gfCNCPoint4[19231] = {X 485.1607, Y 22.5274, Z -6.3333, A 0.000, B 0.000, C 0.000 }
gfCNCPoint4[19232] = {X 489.1455, Y 22.8760, Z -6.3333, A 0.000, B 0.000, C 0.000 }
gfCNCPoint4[19233] = {X 493.6890, Y 22.8760, Z -6.3333, A 0.000, B 0.000, C 0.000 }
gfCNCPoint4[19234] = {X 493.6890, Y 19.4624, Z -6.3333, A 0.000, B 0.000, C 0.000 }
gfCNCPoint4[19235] = {X 487.6634, Y 19.4617, Z -6.3333, A 0.000, B 0.000, C 0.000 }
gfCNCPoint4[19236] = {X 486.9708, Y 19.4665, Z -6.3333, A 0.000, B 0.000, C 0.000 }
gfCNCPoint4[19237] = {X 485.8326, Y 19.5401, Z -6.3333, A 0.000, B 0.000, C 0.000 }
gfCNCPoint4[19238] = {X 484.7145, Y 19.7657, Z -6.3333, A 0.000, B 0.000, C 0.000 }
gfCNCPoint4[19239] = {X 484.4483, Y 19.9152, Z -6.3333, A 0.000, B 0.000, C 0.000 }
gfCNCPoint4[19240] = {X 484.2838, Y 20.1725, Z -6.3333, A 0.000, B 0.000, C 0.000 }
gfCNCPoint4[19241] = {X 484.1061, Y 20.9736, Z -6.3333, A 0.000, B 0.000, C 0.000 }
gfCNCPoint4[19242] = {X 484.1000, Y 21.7941, Z -6.3333, A 0.000, B 0.000, C 0.000 }
gfCNCPoint4[19243] = {X 484.2657, Y 22.5977, Z -6.3333, A 0.000, B 0.000, C 0.000 }
gfCNCPoint4[19244] = {X 484.5770, Y 22.7005, Z -6.3333, A 0.000, B 0.000, C 0.000 }
gfCNCPoint4[19245] = {X 484.9007, Y 22.7530, Z -6.3333, A 0.000, B 0.000, C 0.000 }
gfCNCPoint4[19246] = {X 486.2706, Y 22.8551, Z -6.3333, A 0.000, B 0.000, C 0.000 }
gfCNCPoint4[19247] = {X 487.6442, Y 22.8760, Z -6.3333, A 0.000, B 0.000, C 0.000 }
gfCNCPoint4[19248] = {X 489.1455, Y 22.8760, Z -6.3333, A 0.000, B 0.000, C 0.000 }
gfCNCPoint4[19249] = {X 493.1302, Y 22.5274, Z -6.3333, A 0.000, B 0.000, C 0.000 }
gfCNCPoint4[19250] = {X 485.1607, Y 22.6074, Z -6.3333, A 0.000, B 0.000, C 0.000 }
gfCNCPoint4[19251] = {X 489.1455, Y 22.9560, Z -6.3333, A 0.000, B 0.000, C 0.000 }
gfCNCPoint4[19252] = {X 493.7690, Y 22.9560, Z -6.3333, A 0.000, B 0.000, C 0.000 }
gfCNCPoint4[19253] = {X 493.7690, Y 19.3824, Z -6.3333, A 0.000, B 0.000, C 0.000 }
gfCNCPoint4[19254] = {X 487.6632, Y 19.3817, Z -6.3333, A 0.000, B 0.000, C 0.000 }
gfCNCPoint4[19255] = {X 486.9707, Y 19.3865, Z -6.3333, A 0.000, B 0.000, C 0.000 }
gfCNCPoint4[19256] = {X 485.8219, Y 19.4608, Z -6.3333, A 0.000, B 0.000, C 0.000 }
gfCNCPoint4[19257] = {X 484.6935, Y 19.6886, Z -6.3333, A 0.000, B 0.000, C 0.000 }
gfCNCPoint4[19258] = {X 484.3933, Y 19.8571, Z -6.3333, A 0.000, B 0.000, C 0.000 }
gfCNCPoint4[19259] = {X 484.2079, Y 20.1470, Z -6.3333, A 0.000, B 0.000, C 0.000 }
gfCNCPoint4[19260] = {X 484.0252, Y 20.9767, Z -6.3333, A 0.000, B 0.000, C 0.000 }
gfCNCPoint4[19261] = {X 484.0228, Y 21.8262, Z -6.3333, A 0.000, B 0.000, C 0.000 }
gfCNCPoint4[19262] = {X 484.2007, Y 22.6569, Z -6.3333, A 0.000, B 0.000, C 0.000 }
gfCNCPoint4[19263] = {X 484.5397, Y 22.7736, Z -6.3333, A 0.000, B 0.000, C 0.000 }
gfCNCPoint4[19264] = {X 484.8932, Y 22.8327, Z -6.3333, A 0.000, B 0.000, C 0.000 }
gfCNCPoint4[19265] = {X 486.2672, Y 22.9351, Z -6.3333, A 0.000, B 0.000, C 0.000 }
gfCNCPoint4[19266] = {X 487.6448, Y 22.9560, Z -6.3333, A 0.000, B 0.000, C 0.000 }
gfCNCPoint4[19267] = {X 489.1455, Y 22.9560, Z -6.3333, A 0.000, B 0.000, C 0.000 }
gfCNCPoint4[19268] = {X 493.1302, Y 22.6074, Z -6.3333, A 0.000, B 0.000, C 0.000 }
gfCNCPoint4[19269] = {X 493.1302, Y 22.6074, Z -3.3333, A 0.000, B 0.000, C 0.000 }
gfCNCPoint4[19270] = {X 493.1302, Y 22.6074, Z 11.0000, A 0.000, B 0.000, C 0.000 }
gfCNCPoint4[19271] = {X 448.7147, Y 19.7824, Z 11.0000, A 0.000, B 0.000, C 0.000 }
gfCNCPoint4[19272] = {X 448.7147, Y 19.7824, Z -2.5000, A 0.000, B 0.000, C 0.000 }
gfCNCPoint4[19273] = {X 444.0414, Y 19.7824, Z -3.7522, A 0.000, B 0.000, C 0.000 }
gfCNCPoint4[19274] = {X 443.3486, Y 19.7986, Z -3.9379, A 0.000, B 0.000, C 0.000 }
gfCNCPoint4[19275] = {X 442.7492, Y 19.8053, Z -4.0985, A 0.000, B 0.000, C 0.000 }
gfCNCPoint4[19276] = {X 442.0368, Y 19.9286, Z -4.2922, A 0.000, B 0.000, C 0.000 }
gfCNCPoint4[19277] = {X 441.4699, Y 20.1238, Z -4.4529, A 0.000, B 0.000, C 0.000 }
gfCNCPoint4[19278] = {X 441.3670, Y 20.1592, Z -4.4820, A 0.000, B 0.000, C 0.000 }
gfCNCPoint4[19279] = {X 441.1893, Y 20.7188, Z -4.6394, A 0.000, B 0.000, C 0.000 }
gfCNCPoint4[19280] = {X 441.1557, Y 21.8876, Z -4.9527, A 0.000, B 0.000, C 0.000 }
gfCNCPoint4[19281] = {X 441.2739, Y 22.3510, Z -5.0808, A 0.000, B 0.000, C 0.000 }
gfCNCPoint4[19282] = {X 441.5039, Y 22.4262, Z -5.1457, A 0.000, B 0.000, C 0.000 }
gfCNCPoint4[19283] = {X 441.7450, Y 22.4480, Z -5.2105, A 0.000, B 0.000, C 0.000 }
gfCNCPoint4[19284] = {X 443.0096, Y 22.5623, Z -5.5508, A 0.000, B 0.000, C 0.000 }
gfCNCPoint4[19285] = {X 443.1211, Y 22.5669, Z -5.5807, A 0.000, B 0.000, C 0.000 }
gfCNCPoint4[19286] = {X 444.3942, Y 22.5560, Z -5.9218, A 0.000, B 0.000, C 0.000 }
gfCNCPoint4[19287] = {X 445.9301, Y 22.5560, Z -6.3333, A 0.000, B 0.000, C 0.000 }
gfCNCPoint4[19288] = {X 450.1184, Y 22.5560, Z -6.3333, A 0.000, B 0.000, C 0.000 }
gfCNCPoint4[19289] = {X 450.1184, Y 19.7824, Z -6.3333, A 0.000, B 0.000, C 0.000 }
gfCNCPoint4[19290] = {X 444.0414, Y 19.7824, Z -6.3333, A 0.000, B 0.000, C 0.000 }
gfCNCPoint4[19291] = {X 443.3486, Y 19.7986, Z -6.3333, A 0.000, B 0.000, C 0.000 }
gfCNCPoint4[19292] = {X 442.3962, Y 19.8858, Z -6.3333, A 0.000, B 0.000, C 0.000 }
gfCNCPoint4[19293] = {X 441.4699, Y 20.1238, Z -6.3333, A 0.000, B 0.000, C 0.000 }
gfCNCPoint4[19294] = {X 441.3855, Y 20.1772, Z -6.3333, A 0.000, B 0.000, C 0.000 }
gfCNCPoint4[19295] = {X 441.3341, Y 20.2630, Z -6.3333, A 0.000, B 0.000, C 0.000 }
gfCNCPoint4[19296] = {X 441.1841, Y 20.9512, Z -6.3333, A 0.000, B 0.000, C 0.000 }
gfCNCPoint4[19297] = {X 441.1638, Y 21.6553, Z -6.3333, A 0.000, B 0.000, C 0.000 }
gfCNCPoint4[19298] = {X 441.2739, Y 22.3510, Z -6.3333, A 0.000, B 0.000, C 0.000 }
gfCNCPoint4[19299] = {X 441.5067, Y 22.4128, Z -6.3333, A 0.000, B 0.000, C 0.000 }
gfCNCPoint4[19300] = {X 441.7450, Y 22.4480, Z -6.3333, A 0.000, B 0.000, C 0.000 }
gfCNCPoint4[19301] = {X 443.0683, Y 22.5347, Z -6.3333, A 0.000, B 0.000, C 0.000 }
gfCNCPoint4[19302] = {X 444.3942, Y 22.5560, Z -6.3333, A 0.000, B 0.000, C 0.000 }
gfCNCPoint4[19303] = {X 445.9301, Y 22.5560, Z -6.3333, A 0.000, B 0.000, C 0.000 }
gfCNCPoint4[19304] = {X 441.9453, Y 22.2874, Z -6.3333, A 0.000, B 0.000, C 0.000 }
gfCNCPoint4[19305] = {X 445.9301, Y 22.6360, Z -6.3333, A 0.000, B 0.000, C 0.000 }
gfCNCPoint4[19306] = {X 450.1984, Y 22.6360, Z -6.3333, A 0.000, B 0.000, C 0.000 }
gfCNCPoint4[19307] = {X 450.1984, Y 19.7024, Z -6.3333, A 0.000, B 0.000, C 0.000 }
gfCNCPoint4[19308] = {X 444.0404, Y 19.7024, Z -6.3333, A 0.000, B 0.000, C 0.000 }
gfCNCPoint4[19309] = {X 443.3497, Y 19.7186, Z -6.3333, A 0.000, B 0.000, C 0.000 }
gfCNCPoint4[19310] = {X 442.3835, Y 19.8068, Z -6.3333, A 0.000, B 0.000, C 0.000 }
gfCNCPoint4[19311] = {X 441.4439, Y 20.0481, Z -6.3333, A 0.000, B 0.000, C 0.000 }
gfCNCPoint4[19312] = {X 441.3282, Y 20.1214, Z -6.3333, A 0.000, B 0.000, C 0.000 }
gfCNCPoint4[19313] = {X 441.2578, Y 20.2388, Z -6.3333, A 0.000, B 0.000, C 0.000 }
gfCNCPoint4[19314] = {X 441.1029, Y 20.9559, Z -6.3333, A 0.000, B 0.000, C 0.000 }
gfCNCPoint4[19315] = {X 441.0859, Y 21.6894, Z -6.3333, A 0.000, B 0.000, C 0.000 }
gfCNCPoint4[19316] = {X 441.2074, Y 22.4130, Z -6.3333, A 0.000, B 0.000, C 0.000 }
gfCNCPoint4[19317] = {X 441.4691, Y 22.4867, Z -6.3333, A 0.000, B 0.000, C 0.000 }
gfCNCPoint4[19318] = {X 441.7378, Y 22.5277, Z -6.3333, A 0.000, B 0.000, C 0.000 }
gfCNCPoint4[19319] = {X 443.0640, Y 22.6146, Z -6.3333, A 0.000, B 0.000, C 0.000 }
gfCNCPoint4[19320] = {X 444.3929, Y 22.6360, Z -6.3333, A 0.000, B 0.000, C 0.000 }
gfCNCPoint4[19321] = {X 445.9301, Y 22.6360, Z -6.3333, A 0.000, B 0.000, C 0.000 }
gfCNCPoint4[19322] = {X 449.9148, Y 22.2874, Z -6.3333, A 0.000, B 0.000, C 0.000 }
gfCNCPoint4[19323] = {X 441.9453, Y 22.3674, Z -6.3333, A 0.000, B 0.000, C 0.000 }
gfCNCPoint4[19324] = {X 445.9301, Y 22.7160, Z -6.3333, A 0.000, B 0.000, C 0.000 }
gfCNCPoint4[19325] = {X 450.2784, Y 22.7160, Z -6.3333, A 0.000, B 0.000, C 0.000 }
gfCNCPoint4[19326] = {X 450.2784, Y 19.6224, Z -6.3333, A 0.000, B 0.000, C 0.000 }
gfCNCPoint4[19327] = {X 444.0395, Y 19.6224, Z -6.3333, A 0.000, B 0.000, C 0.000 }
gfCNCPoint4[19328] = {X 443.3483, Y 19.6386, Z -6.3333, A 0.000, B 0.000, C 0.000 }
gfCNCPoint4[19329] = {X 442.3697, Y 19.7280, Z -6.3333, A 0.000, B 0.000, C 0.000 }
gfCNCPoint4[19330] = {X 441.4178, Y 19.9725, Z -6.3333, A 0.000, B 0.000, C 0.000 }
gfCNCPoint4[19331] = {X 441.2710, Y 20.0655, Z -6.3333, A 0.000, B 0.000, C 0.000 }
gfCNCPoint4[19332] = {X 441.1816, Y 20.2145, Z -6.3333, A 0.000, B 0.000, C 0.000 }
gfCNCPoint4[19333] = {X 441.0219, Y 20.9604, Z -6.3333, A 0.000, B 0.000, C 0.000 }
gfCNCPoint4[19334] = {X 441.0082, Y 21.7231, Z -6.3333, A 0.000, B 0.000, C 0.000 }
gfCNCPoint4[19335] = {X 441.1412, Y 22.4742, Z -6.3333, A 0.000, B 0.000, C 0.000 }
gfCNCPoint4[19336] = {X 441.4315, Y 22.5603, Z -6.3333, A 0.000, B 0.000, C 0.000 }
gfCNCPoint4[19337] = {X 441.7306, Y 22.6074, Z -6.3333, A 0.000, B 0.000, C 0.000 }
gfCNCPoint4[19338] = {X 443.0605, Y 22.6946, Z -6.3333, A 0.000, B 0.000, C 0.000 }
gfCNCPoint4[19339] = {X 444.3932, Y 22.7160, Z -6.3333, A 0.000, B 0.000, C 0.000 }
gfCNCPoint4[19340] = {X 445.9301, Y 22.7160, Z -6.3333, A 0.000, B 0.000, C 0.000 }
gfCNCPoint4[19341] = {X 449.9148, Y 22.3674, Z -6.3333, A 0.000, B 0.000, C 0.000 }
gfCNCPoint4[19342] = {X 441.9453, Y 22.4474, Z -6.3333, A 0.000, B 0.000, C 0.000 }
gfCNCPoint4[19343] = {X 445.9301, Y 22.7960, Z -6.3333, A 0.000, B 0.000, C 0.000 }
gfCNCPoint4[19344] = {X 450.3584, Y 22.7960, Z -6.3333, A 0.000, B 0.000, C 0.000 }
gfCNCPoint4[19345] = {X 450.3584, Y 19.5424, Z -6.3333, A 0.000, B 0.000, C 0.000 }
gfCNCPoint4[19346] = {X 444.0385, Y 19.5424, Z -6.3333, A 0.000, B 0.000, C 0.000 }
gfCNCPoint4[19347] = {X 443.3469, Y 19.5586, Z -6.3333, A 0.000, B 0.000, C 0.000 }
gfCNCPoint4[19348] = {X 442.3558, Y 19.6492, Z -6.3333, A 0.000, B 0.000, C 0.000 }
gfCNCPoint4[19349] = {X 441.3918, Y 19.8968, Z -6.3333, A 0.000, B 0.000, C 0.000 }
gfCNCPoint4[19350] = {X 441.2137, Y 20.0096, Z -6.3333, A 0.000, B 0.000, C 0.000 }
gfCNCPoint4[19351] = {X 441.1053, Y 20.1903, Z -6.3333, A 0.000, B 0.000, C 0.000 }
gfCNCPoint4[19352] = {X 440.9409, Y 20.9647, Z -6.3333, A 0.000, B 0.000, C 0.000 }
gfCNCPoint4[19353] = {X 440.9307, Y 21.7563, Z -6.3333, A 0.000, B 0.000, C 0.000 }
gfCNCPoint4[19354] = {X 441.0752, Y 22.5347, Z -6.3333, A 0.000, B 0.000, C 0.000 }
gfCNCPoint4[19355] = {X 441.3939, Y 22.6337, Z -6.3333, A 0.000, B 0.000, C 0.000 }
gfCNCPoint4[19356] = {X 441.7233, Y 22.6870, Z -6.3333, A 0.000, B 0.000, C 0.000 }
gfCNCPoint4[19357] = {X 443.0571, Y 22.7745, Z -6.3333, A 0.000, B 0.000, C 0.000 }
gfCNCPoint4[19358] = {X 444.3936, Y 22.7960, Z -6.3333, A 0.000, B 0.000, C 0.000 }
gfCNCPoint4[19359] = {X 445.9301, Y 22.7960, Z -6.3333, A 0.000, B 0.000, C 0.000 }
gfCNCPoint4[19360] = {X 449.9148, Y 22.4474, Z -6.3333, A 0.000, B 0.000, C 0.000 }
gfCNCPoint4[19361] = {X 441.9453, Y 22.5274, Z -6.3333, A 0.000, B 0.000, C 0.000 }
gfCNCPoint4[19362] = {X 445.9301, Y 22.8760, Z -6.3333, A 0.000, B 0.000, C 0.000 }
gfCNCPoint4[19363] = {X 450.4384, Y 22.8760, Z -6.3333, A 0.000, B 0.000, C 0.000 }
gfCNCPoint4[19364] = {X 450.4384, Y 19.4624, Z -6.3333, A 0.000, B 0.000, C 0.000 }
gfCNCPoint4[19365] = {X 444.0376, Y 19.4624, Z -6.3333, A 0.000, B 0.000, C 0.000 }
gfCNCPoint4[19366] = {X 443.3456, Y 19.4786, Z -6.3333, A 0.000, B 0.000, C 0.000 }
gfCNCPoint4[19367] = {X 442.3419, Y 19.5704, Z -6.3333, A 0.000, B 0.000, C 0.000 }
gfCNCPoint4[19368] = {X 441.3658, Y 19.8212, Z -6.3333, A 0.000, B 0.000, C 0.000 }
gfCNCPoint4[19369] = {X 441.1565, Y 19.9537, Z -6.3333, A 0.000, B 0.000, C 0.000 }
gfCNCPoint4[19370] = {X 441.0291, Y 20.1661, Z -6.3333, A 0.000, B 0.000, C 0.000 }
gfCNCPoint4[19371] = {X 440.8599, Y 20.9689, Z -6.3333, A 0.000, B 0.000, C 0.000 }
gfCNCPoint4[19372] = {X 440.8533, Y 21.7892, Z -6.3333, A 0.000, B 0.000, C 0.000 }
gfCNCPoint4[19373] = {X 441.0095, Y 22.5946, Z -6.3333, A 0.000, B 0.000, C 0.000 }
gfCNCPoint4[19374] = {X 441.3564, Y 22.7070, Z -6.3333, A 0.000, B 0.000, C 0.000 }
gfCNCPoint4[19375] = {X 441.7161, Y 22.7667, Z -6.3333, A 0.000, B 0.000, C 0.000 }
gfCNCPoint4[19376] = {X 443.0537, Y 22.8544, Z -6.3333, A 0.000, B 0.000, C 0.000 }
gfCNCPoint4[19377] = {X 444.3939, Y 22.8760, Z -6.3333, A 0.000, B 0.000, C 0.000 }
gfCNCPoint4[19378] = {X 445.9301, Y 22.8760, Z -6.3333, A 0.000, B 0.000, C 0.000 }
gfCNCPoint4[19379] = {X 449.9148, Y 22.5274, Z -6.3333, A 0.000, B 0.000, C 0.000 }
gfCNCPoint4[19380] = {X 441.9453, Y 22.6074, Z -6.3333, A 0.000, B 0.000, C 0.000 }
gfCNCPoint4[19381] = {X 445.9301, Y 22.9560, Z -6.3333, A 0.000, B 0.000, C 0.000 }
gfCNCPoint4[19382] = {X 450.5184, Y 22.9560, Z -6.3333, A 0.000, B 0.000, C 0.000 }
gfCNCPoint4[19383] = {X 450.5185, Y 19.3824, Z -6.3333, A 0.000, B 0.000, C 0.000 }
gfCNCPoint4[19384] = {X 444.0367, Y 19.3824, Z -6.3333, A 0.000, B 0.000, C 0.000 }
gfCNCPoint4[19385] = {X 443.3442, Y 19.3987, Z -6.3333, A 0.000, B 0.000, C 0.000 }
gfCNCPoint4[19386] = {X 442.3280, Y 19.4916, Z -6.3333, A 0.000, B 0.000, C 0.000 }
gfCNCPoint4[19387] = {X 441.3397, Y 19.7456, Z -6.3333, A 0.000, B 0.000, C 0.000 }
gfCNCPoint4[19388] = {X 441.0992, Y 19.8978, Z -6.3333, A 0.000, B 0.000, C 0.000 }
gfCNCPoint4[19389] = {X 440.9528, Y 20.1419, Z -6.3333, A 0.000, B 0.000, C 0.000 }
gfCNCPoint4[19390] = {X 440.7791, Y 20.9729, Z -6.3333, A 0.000, B 0.000, C 0.000 }
gfCNCPoint4[19391] = {X 440.7761, Y 21.8218, Z -6.3333, A 0.000, B 0.000, C 0.000 }
gfCNCPoint4[19392] = {X 440.9439, Y 22.6539, Z -6.3333, A 0.000, B 0.000, C 0.000 }
gfCNCPoint4[19393] = {X 441.3189, Y 22.7801, Z -6.3333, A 0.000, B 0.000, C 0.000 }
gfCNCPoint4[19394] = {X 441.7090, Y 22.8464, Z -6.3333, A 0.000, B 0.000, C 0.000 }
gfCNCPoint4[19395] = {X 443.0503, Y 22.9343, Z -6.3333, A 0.000, B 0.000, C 0.000 }
gfCNCPoint4[19396] = {X 444.3942, Y 22.9560, Z -6.3333, A 0.000, B 0.000, C 0.000 }
gfCNCPoint4[19397] = {X 445.9301, Y 22.9560, Z -6.3333, A 0.000, B 0.000, C 0.000 }
gfCNCPoint4[19398] = {X 449.9301, Y 22.9560, Z -6.3333, A 0.000, B 0.000, C 0.000 }
gfCNCPoint4[19399] = {X 449.9301, Y 22.9560, Z -3.3333, A 0.000, B 0.000, C 0.000 }
gfCNCPoint4[19400] = {X 449.9301, Y 22.9560, Z 11.0000, A 0.000, B 0.000, C 0.000 }
gfCNCPoint4[19401] = {X 507.6813, Y 107.6951, Z 11.0000, A 0.000, B 0.000, C 0.000 }
gfCNCPoint4[19402] = {X 507.6813, Y 107.6951, Z -3.3333, A 0.000, B 0.000, C 0.000 }
gfCNCPoint4[19403] = {X 507.6813, Y 107.6951, Z -6.3333, A 0.000, B 0.000, C 0.000 }
gfCNCPoint4[19404] = {X 507.6813, Y 71.2951, Z -6.3333, A 0.000, B 0.000, C 0.000 }
gfCNCPoint4[19405] = {X 509.5504, Y 71.2951, Z -6.3333, A 0.000, B 0.000, C 0.000 }
gfCNCPoint4[19406] = {X 509.0279, Y 71.0692, Z -6.3333, A 0.000, B 0.000, C 0.000 }
gfCNCPoint4[19407] = {X 508.5105, Y 70.8320, Z -6.3333, A 0.000, B 0.000, C 0.000 }
gfCNCPoint4[19408] = {X 507.1674, Y 71.0985, Z -6.3333, A 0.000, B 0.000, C 0.000 }
gfCNCPoint4[19409] = {X 505.8123, Y 71.2951, Z -6.3333, A 0.000, B 0.000, C 0.000 }
gfCNCPoint4[19410] = {X 507.6813, Y 71.2951, Z -6.3333, A 0.000, B 0.000, C 0.000 }
gfCNCPoint4[19411] = {X 507.6813, Y 73.6951, Z -6.3333, A 0.000, B 0.000, C 0.000 }
gfCNCPoint4[19412] = {X 551.2536, Y 73.6951, Z -6.3333, A 0.000, B 0.000, C 0.000 }
gfCNCPoint4[19413] = {X 549.1242, Y 72.7707, Z -6.3333, A 0.000, B 0.000, C 0.000 }
gfCNCPoint4[19414] = {X 547.0704, Y 71.6886, Z -6.3333, A 0.000, B 0.000, C 0.000 }
gfCNCPoint4[19415] = {X 545.1040, Y 70.4549, Z -6.3333, A 0.000, B 0.000, C 0.000 }
gfCNCPoint4[19416] = {X 543.2360, Y 69.0766, Z -6.3333, A 0.000, B 0.000, C 0.000 }
gfCNCPoint4[19417] = {X 529.7629, Y 69.0769, Z -6.3333, A 0.000, B 0.000, C 0.000 }
gfCNCPoint4[19418] = {X 527.5492, Y 69.8803, Z -6.3333, A 0.000, B 0.000, C 0.000 }
gfCNCPoint4[19419] = {X 525.2680, Y 70.4651, Z -6.3333, A 0.000, B 0.000, C 0.000 }
gfCNCPoint4[19420] = {X 522.9408, Y 70.8258, Z -6.3333, A 0.000, B 0.000, C 0.000 }
gfCNCPoint4[19421] = {X 520.5895, Y 70.9589, Z -6.3333, A 0.000, B 0.000, C 0.000 }
gfCNCPoint4[19422] = {X 519.7998, Y 70.9591, Z -6.3333, A 0.000, B 0.000, C 0.000 }
gfCNCPoint4[19423] = {X 517.4111, Y 70.8404, Z -6.3333, A 0.000, B 0.000, C 0.000 }
gfCNCPoint4[19424] = {X 515.0460, Y 70.4852, Z -6.3333, A 0.000, B 0.000, C 0.000 }
gfCNCPoint4[19425] = {X 512.7278, Y 69.8972, Z -6.3333, A 0.000, B 0.000, C 0.000 }
gfCNCPoint4[19426] = {X 510.4793, Y 69.0822, Z -6.3333, A 0.000, B 0.000, C 0.000 }
gfCNCPoint4[19427] = {X 509.6266, Y 68.7046, Z -6.3333, A 0.000, B 0.000, C 0.000 }
gfCNCPoint4[19428] = {X 508.7892, Y 68.2944, Z -6.3333, A 0.000, B 0.000, C 0.000 }
gfCNCPoint4[19429] = {X 507.1698, Y 68.6593, Z -6.3333, A 0.000, B 0.000, C 0.000 }
gfCNCPoint4[19430] = {X 505.5292, Y 68.9119, Z -6.3333, A 0.000, B 0.000, C 0.000 }
gfCNCPoint4[19431] = {X 504.1113, Y 69.0379, Z -6.3333, A 0.000, B 0.000, C 0.000 }
gfCNCPoint4[19432] = {X 502.6885, Y 69.0800, Z -6.3333, A 0.000, B 0.000, C 0.000 }
gfCNCPoint4[19433] = {X 502.0391, Y 69.0800, Z -6.3333, A 0.000, B 0.000, C 0.000 }
gfCNCPoint4[19434] = {X 501.1777, Y 71.1317, Z -6.3333, A 0.000, B 0.000, C 0.000 }
gfCNCPoint4[19435] = {X 500.1609, Y 73.1110, Z -6.3333, A 0.000, B 0.000, C 0.000 }
gfCNCPoint4[19436] = {X 500.1609, Y 73.6951, Z -6.3333, A 0.000, B 0.000, C 0.000 }
gfCNCPoint4[19437] = {X 507.6813, Y 73.6951, Z -6.3333, A 0.000, B 0.000, C 0.000 }
gfCNCPoint4[19438] = {X 507.6813, Y 76.0951, Z -6.3333, A 0.000, B 0.000, C 0.000 }
gfCNCPoint4[19439] = {X 576.0966, Y 76.0951, Z -6.3333, A 0.000, B 0.000, C 0.000 }
gfCNCPoint4[19440] = {X 576.0966, Y 72.8901, Z -6.3333, A 0.000, B 0.000, C 0.000 }
gfCNCPoint4[19441] = {X 575.7179, Y 72.8147, Z -6.3333, A 0.000, B 0.000, C 0.000 }
gfCNCPoint4[19442] = {X 575.3401, Y 72.7341, Z -6.3333, A 0.000, B 0.000, C 0.000 }
gfCNCPoint4[19443] = {X 573.3201, Y 73.1034, Z -6.3333, A 0.000, B 0.000, C 0.000 }
gfCNCPoint4[19444] = {X 571.2786, Y 73.3258, Z -6.3333, A 0.000, B 0.000, C 0.000 }
gfCNCPoint4[19445] = {X 569.2264, Y 73.4000, Z -6.3333, A 0.000, B 0.000, C 0.000 }
gfCNCPoint4[19446] = {X 562.4443, Y 73.4000, Z -6.3333, A 0.000, B 0.000, C 0.000 }
gfCNCPoint4[19447] = {X 560.3342, Y 73.3215, Z -6.3333, A 0.000, B 0.000, C 0.000 }
gfCNCPoint4[19448] = {X 558.2357, Y 73.0864, Z -6.3333, A 0.000, B 0.000, C 0.000 }
gfCNCPoint4[19449] = {X 556.1605, Y 72.6961, Z -6.3333, A 0.000, B 0.000, C 0.000 }
gfCNCPoint4[19450] = {X 554.1201, Y 72.1527, Z -6.3333, A 0.000, B 0.000, C 0.000 }
gfCNCPoint4[19451] = {X 552.1256, Y 71.4591, Z -6.3333, A 0.000, B 0.000, C 0.000 }
gfCNCPoint4[19452] = {X 549.9766, Y 70.5170, Z -6.3333, A 0.000, B 0.000, C 0.000 }
gfCNCPoint4[19453] = {X 547.9126, Y 69.4006, Z -6.3333, A 0.000, B 0.000, C 0.000 }
gfCNCPoint4[19454] = {X 545.9479, Y 68.1177, Z -6.3333, A 0.000, B 0.000, C 0.000 }
gfCNCPoint4[19455] = {X 544.0958, Y 66.6770, Z -6.3333, A 0.000, B 0.000, C 0.000 }
gfCNCPoint4[19456] = {X 543.8504, Y 66.6782, Z -6.3333, A 0.000, B 0.000, C 0.000 }
gfCNCPoint4[19457] = {X 543.6050, Y 66.6766, Z -6.3333, A 0.000, B 0.000, C 0.000 }
gfCNCPoint4[19458] = {X 529.2673, Y 66.6769, Z -6.3333, A 0.000, B 0.000, C 0.000 }
gfCNCPoint4[19459] = {X 527.1772, Y 67.4804, Z -6.3333, A 0.000, B 0.000, C 0.000 }
gfCNCPoint4[19460] = {X 525.0157, Y 68.0656, Z -6.3333, A 0.000, B 0.000, C 0.000 }
gfCNCPoint4[19461] = {X 522.8057, Y 68.4264, Z -6.3333, A 0.000, B 0.000, C 0.000 }
gfCNCPoint4[19462] = {X 520.5703, Y 68.5590, Z -6.3333, A 0.000, B 0.000, C 0.000 }
gfCNCPoint4[19463] = {X 519.7998, Y 68.5591, Z -6.3333, A 0.000, B 0.000, C 0.000 }
gfCNCPoint4[19464] = {X 517.5593, Y 68.4430, Z -6.3333, A 0.000, B 0.000, C 0.000 }
gfCNCPoint4[19465] = {X 515.3429, Y 68.0961, Z -6.3333, A 0.000, B 0.000, C 0.000 }
gfCNCPoint4[19466] = {X 513.1742, Y 67.5219, Z -6.3333, A 0.000, B 0.000, C 0.000 }
gfCNCPoint4[19467] = {X 511.0764, Y 66.7267, Z -6.3333, A 0.000, B 0.000, C 0.000 }
gfCNCPoint4[19468] = {X 509.0720, Y 65.7189, Z -6.3333, A 0.000, B 0.000, C 0.000 }
gfCNCPoint4[19469] = {X 506.9797, Y 66.2511, Z -6.3333, A 0.000, B 0.000, C 0.000 }
gfCNCPoint4[19470] = {X 504.8448, Y 66.5725, Z -6.3333, A 0.000, B 0.000, C 0.000 }
gfCNCPoint4[19471] = {X 502.6885, Y 66.6800, Z -6.3333, A 0.000, B 0.000, C 0.000 }
gfCNCPoint4[19472] = {X 500.3217, Y 66.6800, Z -6.3333, A 0.000, B 0.000, C 0.000 }
gfCNCPoint4[19473] = {X 499.6232, Y 68.6751, Z -6.3333, A 0.000, B 0.000, C 0.000 }
gfCNCPoint4[19474] = {X 498.7678, Y 70.6081, Z -6.3333, A 0.000, B 0.000, C 0.000 }
gfCNCPoint4[19475] = {X 497.7609, Y 72.4667, Z -6.3333, A 0.000, B 0.000, C 0.000 }
gfCNCPoint4[19476] = {X 497.7609, Y 76.0951, Z -6.3333, A 0.000, B 0.000, C 0.000 }
gfCNCPoint4[19477] = {X 507.6813, Y 76.0951, Z -6.3333, A 0.000, B 0.000, C 0.000 }
gfCNCPoint4[19478] = {X 507.6813, Y 78.4951, Z -6.3333, A 0.000, B 0.000, C 0.000 }
gfCNCPoint4[19479] = {X 578.4966, Y 78.4951, Z -6.3333, A 0.000, B 0.000, C 0.000 }
gfCNCPoint4[19480] = {X 578.4966, Y 70.8313, Z -6.3333, A 0.000, B 0.000, C 0.000 }
gfCNCPoint4[19481] = {X 576.9097, Y 70.5998, Z -6.3333, A 0.000, B 0.000, C 0.000 }
gfCNCPoint4[19482] = {X 575.3401, Y 70.2710, Z -6.3333, A 0.000, B 0.000, C 0.000 }
gfCNCPoint4[19483] = {X 573.3236, Y 70.6751, Z -6.3333, A 0.000, B 0.000, C 0.000 }
gfCNCPoint4[19484] = {X 571.2815, Y 70.9187, Z -6.3333, A 0.000, B 0.000, C 0.000 }
gfCNCPoint4[19485] = {X 569.2264, Y 71.0000, Z -6.3333, A 0.000, B 0.000, C 0.000 }
gfCNCPoint4[19486] = {X 562.4443, Y 71.0000, Z -6.3333, A 0.000, B 0.000, C 0.000 }
gfCNCPoint4[19487] = {X 560.1227, Y 70.8961, Z -6.3333, A 0.000, B 0.000, C 0.000 }
gfCNCPoint4[19488] = {X 557.8196, Y 70.5854, Z -6.3333, A 0.000, B 0.000, C 0.000 }
gfCNCPoint4[19489] = {X 555.5535, Y 70.0702, Z -6.3333, A 0.000, B 0.000, C 0.000 }
gfCNCPoint4[19490] = {X 553.3425, Y 69.3548, Z -6.3333, A 0.000, B 0.000, C 0.000 }
gfCNCPoint4[19491] = {X 551.2041, Y 68.4448, Z -6.3333, A 0.000, B 0.000, C 0.000 }
gfCNCPoint4[19492] = {X 549.1556, Y 67.3475, Z -6.3333, A 0.000, B 0.000, C 0.000 }
gfCNCPoint4[19493] = {X 547.2132, Y 66.0716, Z -6.3333, A 0.000, B 0.000, C 0.000 }
gfCNCPoint4[19494] = {X 545.3925, Y 64.6274, Z -6.3333, A 0.000, B 0.000, C 0.000 }
gfCNCPoint4[19495] = {X 545.1773, Y 64.4384, Z -6.3333, A 0.000, B 0.000, C 0.000 }
gfCNCPoint4[19496] = {X 544.9642, Y 64.2469, Z -6.3333, A 0.000, B 0.000, C 0.000 }
gfCNCPoint4[19497] = {X 544.2923, Y 64.2735, Z -6.3333, A 0.000, B 0.000, C 0.000 }
gfCNCPoint4[19498] = {X 543.6199, Y 64.2766, Z -6.3333, A 0.000, B 0.000, C 0.000 }
gfCNCPoint4[19499] = {X 528.7423, Y 64.2769, Z -6.3333, A 0.000, B 0.000, C 0.000 }
gfCNCPoint4[19500] = {X 526.7860, Y 65.0796, Z -6.3333, A 0.000, B 0.000, C 0.000 }
gfCNCPoint4[19501] = {X 524.7540, Y 65.6650, Z -6.3333, A 0.000, B 0.000, C 0.000 }
gfCNCPoint4[19502] = {X 522.6705, Y 66.0262, Z -6.3333, A 0.000, B 0.000, C 0.000 }
gfCNCPoint4[19503] = {X 520.5601, Y 66.1590, Z -6.3333, A 0.000, B 0.000, C 0.000 }
gfCNCPoint4[19504] = {X 519.7998, Y 66.1591, Z -6.3333, A 0.000, B 0.000, C 0.000 }
gfCNCPoint4[19505] = {X 517.9641, Y 66.0715, Z -6.3333, A 0.000, B 0.000, C 0.000 }
gfCNCPoint4[19506] = {X 516.1450, Y 65.8096, Z -6.3333, A 0.000, B 0.000, C 0.000 }
gfCNCPoint4[19507] = {X 514.3592, Y 65.3756, Z -6.3333, A 0.000, B 0.000, C 0.000 }
gfCNCPoint4[19508] = {X 512.6228, Y 64.7735, Z -6.3333, A 0.000, B 0.000, C 0.000 }
gfCNCPoint4[19509] = {X 510.9516, Y 64.0089, Z -6.3333, A 0.000, B 0.000, C 0.000 }
gfCNCPoint4[19510] = {X 509.3609, Y 63.0886, Z -6.3333, A 0.000, B 0.000, C 0.000 }
gfCNCPoint4[19511] = {X 507.7389, Y 63.6068, Z -6.3333, A 0.000, B 0.000, C 0.000 }
gfCNCPoint4[19512] = {X 506.0774, Y 63.9798, Z -6.3333, A 0.000, B 0.000, C 0.000 }
gfCNCPoint4[19513] = {X 504.3896, Y 64.2048, Z -6.3333, A 0.000, B 0.000, C 0.000 }
gfCNCPoint4[19514] = {X 502.6885, Y 64.2800, Z -6.3333, A 0.000, B 0.000, C 0.000 }
gfCNCPoint4[19515] = {X 498.4791, Y 64.2800, Z -6.3333, A 0.000, B 0.000, C 0.000 }
gfCNCPoint4[19516] = {X 497.9417, Y 66.2502, Z -6.3333, A 0.000, B 0.000, C 0.000 }
gfCNCPoint4[19517] = {X 497.2393, Y 68.1677, Z -6.3333, A 0.000, B 0.000, C 0.000 }
gfCNCPoint4[19518] = {X 496.3769, Y 70.0188, Z -6.3333, A 0.000, B 0.000, C 0.000 }
gfCNCPoint4[19519] = {X 495.3609, Y 71.7903, Z -6.3333, A 0.000, B 0.000, C 0.000 }
gfCNCPoint4[19520] = {X 495.3610, Y 78.4951, Z -6.3333, A 0.000, B 0.000, C 0.000 }
gfCNCPoint4[19521] = {X 507.6813, Y 78.4951, Z -6.3333, A 0.000, B 0.000, C 0.000 }
gfCNCPoint4[19522] = {X 507.6813, Y 80.8951, Z -6.3333, A 0.000, B 0.000, C 0.000 }
gfCNCPoint4[19523] = {X 580.8966, Y 80.8951, Z -6.3333, A 0.000, B 0.000, C 0.000 }
gfCNCPoint4[19524] = {X 580.8966, Y 68.5934, Z -6.3333, A 0.000, B 0.000, C 0.000 }
gfCNCPoint4[19525] = {X 579.0252, Y 68.4747, Z -6.3333, A 0.000, B 0.000, C 0.000 }
gfCNCPoint4[19526] = {X 577.1692, Y 68.2078, Z -6.3333, A 0.000, B 0.000, C 0.000 }
gfCNCPoint4[19527] = {X 575.3401, Y 67.7943, Z -6.3333, A 0.000, B 0.000, C 0.000 }
gfCNCPoint4[19528] = {X 573.3283, Y 68.2408, Z -6.3333, A 0.000, B 0.000, C 0.000 }
gfCNCPoint4[19529] = {X 571.2852, Y 68.5100, Z -6.3333, A 0.000, B 0.000, C 0.000 }
gfCNCPoint4[19530] = {X 569.2264, Y 68.6000, Z -6.3333, A 0.000, B 0.000, C 0.000 }
gfCNCPoint4[19531] = {X 562.4443, Y 68.6000, Z -6.3333, A 0.000, B 0.000, C 0.000 }
gfCNCPoint4[19532] = {X 560.3370, Y 68.5057, Z -6.3333, A 0.000, B 0.000, C 0.000 }
gfCNCPoint4[19533] = {X 558.2465, Y 68.2237, Z -6.3333, A 0.000, B 0.000, C 0.000 }
gfCNCPoint4[19534] = {X 556.1896, Y 67.7561, Z -6.3333, A 0.000, B 0.000, C 0.000 }
gfCNCPoint4[19535] = {X 554.1826, Y 67.1067, Z -6.3333, A 0.000, B 0.000, C 0.000 }
gfCNCPoint4[19536] = {X 552.2417, Y 66.2807, Z -6.3333, A 0.000, B 0.000, C 0.000 }
gfCNCPoint4[19537] = {X 550.3822, Y 65.2846, Z -6.3333, A 0.000, B 0.000, C 0.000 }
gfCNCPoint4[19538] = {X 548.6191, Y 64.1265, Z -6.3333, A 0.000, B 0.000, C 0.000 }
gfCNCPoint4[19539] = {X 546.9665, Y 62.8157, Z -6.3333, A 0.000, B 0.000, C 0.000 }
gfCNCPoint4[19540] = {X 546.3909, Y 62.2988, Z -6.3333, A 0.000, B 0.000, C 0.000 }
gfCNCPoint4[19541] = {X 545.8326, Y 61.7634, Z -6.3333, A 0.000, B 0.000, C 0.000 }
gfCNCPoint4[19542] = {X 544.7360, Y 61.8558, Z -6.3333, A 0.000, B 0.000, C 0.000 }
gfCNCPoint4[19543] = {X 543.6358, Y 61.8766, Z -6.3333, A 0.000, B 0.000, C 0.000 }
gfCNCPoint4[19544] = {X 528.1820, Y 61.8769, Z -6.3333, A 0.000, B 0.000, C 0.000 }
gfCNCPoint4[19545] = {X 526.3693, Y 62.6785, Z -6.3333, A 0.000, B 0.000, C 0.000 }
gfCNCPoint4[19546] = {X 524.4756, Y 63.2642, Z -6.3333, A 0.000, B 0.000, C 0.000 }
gfCNCPoint4[19547] = {X 522.5268, Y 63.6260, Z -6.3333, A 0.000, B 0.000, C 0.000 }
gfCNCPoint4[19548] = {X 520.5491, Y 63.7590, Z -6.3333, A 0.000, B 0.000, C 0.000 }
gfCNCPoint4[19549] = {X 519.7998, Y 63.7591, Z -6.3333, A 0.000, B 0.000, C 0.000 }
gfCNCPoint4[19550] = {X 517.9902, Y 63.6618, Z -6.3333, A 0.000, B 0.000, C 0.000 }
gfCNCPoint4[19551] = {X 516.2015, Y 63.3711, Z -6.3333, A 0.000, B 0.000, C 0.000 }
gfCNCPoint4[19552] = {X 514.4543, Y 62.8904, Z -6.3333, A 0.000, B 0.000, C 0.000 }
gfCNCPoint4[19553] = {X 512.7687, Y 62.2251, Z -6.3333, A 0.000, B 0.000, C 0.000 }
gfCNCPoint4[19554] = {X 511.1641, Y 61.3829, Z -6.3333, A 0.000, B 0.000, C 0.000 }
gfCNCPoint4[19555] = {X 509.6590, Y 60.3735, Z -6.3333, A 0.000, B 0.000, C 0.000 }
gfCNCPoint4[19556] = {X 507.9866, Y 61.0270, Z -6.3333, A 0.000, B 0.000, C 0.000 }
gfCNCPoint4[19557] = {X 506.2542, Y 61.4991, Z -6.3333, A 0.000, B 0.000, C 0.000 }
gfCNCPoint4[19558] = {X 504.4815, Y 61.7845, Z -6.3333, A 0.000, B 0.000, C 0.000 }
gfCNCPoint4[19559] = {X 502.6885, Y 61.8800, Z -6.3333, A 0.000, B 0.000, C 0.000 }
gfCNCPoint4[19560] = {X 496.4789, Y 61.8800, Z -6.3333, A 0.000, B 0.000, C 0.000 }
gfCNCPoint4[19561] = {X 496.1192, Y 63.8330, Z -6.3333, A 0.000, B 0.000, C 0.000 }
gfCNCPoint4[19562] = {X 495.5824, Y 65.7449, Z -6.3333, A 0.000, B 0.000, C 0.000 }
gfCNCPoint4[19563] = {X 494.8728, Y 67.5997, Z -6.3333, A 0.000, B 0.000, C 0.000 }
gfCNCPoint4[19564] = {X 493.9965, Y 69.3817, Z -6.3333, A 0.000, B 0.000, C 0.000 }
gfCNCPoint4[19565] = {X 492.9608, Y 71.0761, Z -6.3333, A 0.000, B 0.000, C 0.000 }
gfCNCPoint4[19566] = {X 492.9610, Y 80.8951, Z -6.3333, A 0.000, B 0.000, C 0.000 }
gfCNCPoint4[19567] = {X 507.6813, Y 80.8951, Z -6.3333, A 0.000, B 0.000, C 0.000 }
gfCNCPoint4[19568] = {X 507.6813, Y 83.2951, Z -6.3333, A 0.000, B 0.000, C 0.000 }
gfCNCPoint4[19569] = {X 583.2966, Y 83.2951, Z -6.3333, A 0.000, B 0.000, C 0.000 }
gfCNCPoint4[19570] = {X 583.2966, Y 66.1198, Z -6.3333, A 0.000, B 0.000, C 0.000 }
gfCNCPoint4[19571] = {X 581.2872, Y 66.1993, Z -6.3333, A 0.000, B 0.000, C 0.000 }
gfCNCPoint4[19572] = {X 579.2793, Y 66.0882, Z -6.3333, A 0.000, B 0.000, C 0.000 }
gfCNCPoint4[19573] = {X 577.2910, Y 65.7873, Z -6.3333, A 0.000, B 0.000, C 0.000 }
gfCNCPoint4[19574] = {X 575.3401, Y 65.2993, Z -6.3333, A 0.000, B 0.000, C 0.000 }
gfCNCPoint4[19575] = {X 573.3348, Y 65.7981, Z -6.3333, A 0.000, B 0.000, C 0.000 }
gfCNCPoint4[19576] = {X 571.2904, Y 66.0993, Z -6.3333, A 0.000, B 0.000, C 0.000 }
gfCNCPoint4[19577] = {X 569.2264, Y 66.2000, Z -6.3333, A 0.000, B 0.000, C 0.000 }
gfCNCPoint4[19578] = {X 562.4443, Y 66.2000, Z -6.3333, A 0.000, B 0.000, C 0.000 }
gfCNCPoint4[19579] = {X 560.2817, Y 66.0894, Z -6.3333, A 0.000, B 0.000, C 0.000 }
gfCNCPoint4[19580] = {X 558.1418, Y 65.7588, Z -6.3333, A 0.000, B 0.000, C 0.000 }
gfCNCPoint4[19581] = {X 556.0467, Y 65.2116, Z -6.3333, A 0.000, B 0.000, C 0.000 }
gfCNCPoint4[19582] = {X 554.0183, Y 64.4536, Z -6.3333, A 0.000, B 0.000, C 0.000 }
gfCNCPoint4[19583] = {X 552.0779, Y 63.4926, Z -6.3333, A 0.000, B 0.000, C 0.000 }
gfCNCPoint4[19584] = {X 550.2455, Y 62.3387, Z -6.3333, A 0.000, B 0.000, C 0.000 }
gfCNCPoint4[19585] = {X 548.5405, Y 61.0039, Z -6.3333, A 0.000, B 0.000, C 0.000 }
gfCNCPoint4[19586] = {X 547.5933, Y 60.1290, Z -6.3333, A 0.000, B 0.000, C 0.000 }
gfCNCPoint4[19587] = {X 546.7010, Y 59.1982, Z -6.3333, A 0.000, B 0.000, C 0.000 }
gfCNCPoint4[19588] = {X 545.1843, Y 59.4182, Z -6.3333, A 0.000, B 0.000, C 0.000 }
gfCNCPoint4[19589] = {X 543.6528, Y 59.4766, Z -6.3333, A 0.000, B 0.000, C 0.000 }
gfCNCPoint4[19590] = {X 527.5782, Y 59.4769, Z -6.3333, A 0.000, B 0.000, C 0.000 }
gfCNCPoint4[19591] = {X 525.9211, Y 60.2772, Z -6.3333, A 0.000, B 0.000, C 0.000 }
gfCNCPoint4[19592] = {X 524.1768, Y 60.8632, Z -6.3333, A 0.000, B 0.000, C 0.000 }
gfCNCPoint4[19593] = {X 522.3727, Y 61.2257, Z -6.3333, A 0.000, B 0.000, C 0.000 }
gfCNCPoint4[19594] = {X 520.5374, Y 61.3590, Z -6.3333, A 0.000, B 0.000, C 0.000 }
gfCNCPoint4[19595] = {X 519.7998, Y 61.3591, Z -6.3333, A 0.000, B 0.000, C 0.000 }
gfCNCPoint4[19596] = {X 518.0043, Y 61.2474, Z -6.3333, A 0.000, B 0.000, C 0.000 }
gfCNCPoint4[19597] = {X 516.2365, Y 60.9138, Z -6.3333, A 0.000, B 0.000, C 0.000 }
gfCNCPoint4[19598] = {X 514.5237, Y 60.3637, Z -6.3333, A 0.000, B 0.000, C 0.000 }
gfCNCPoint4[19599] = {X 512.8923, Y 59.6054, Z -6.3333, A 0.000, B 0.000, C 0.000 }
gfCNCPoint4[19600] = {X 511.3676, Y 58.6507, Z -6.3333, A 0.000, B 0.000, C 0.000 }
gfCNCPoint4[19601] = {X 509.9730, Y 57.5142, Z -6.3333, A 0.000, B 0.000, C 0.000 }
gfCNCPoint4[19602] = {X 508.6156, Y 58.2113, Z -6.3333, A 0.000, B 0.000, C 0.000 }
gfCNCPoint4[19603] = {X 507.1924, Y 58.7617, Z -6.3333, A 0.000, B 0.000, C 0.000 }
gfCNCPoint4[19604] = {X 505.7192, Y 59.1593, Z -6.3333, A 0.000, B 0.000, C 0.000 }
gfCNCPoint4[19605] = {X 504.2123, Y 59.3996, Z -6.3333, A 0.000, B 0.000, C 0.000 }
gfCNCPoint4[19606] = {X 502.6885, Y 59.4800, Z -6.3333, A 0.000, B 0.000, C 0.000 }
gfCNCPoint4[19607] = {X 496.2450, Y 59.4800, Z -6.3333, A 0.000, B 0.000, C 0.000 }
gfCNCPoint4[19608] = {X 495.2580, Y 59.4463, Z -6.3333, A 0.000, B 0.000, C 0.000 }
gfCNCPoint4[19609] = {X 494.2756, Y 59.3454, Z -6.3333, A 0.000, B 0.000, C 0.000 }
gfCNCPoint4[19610] = {X 494.1342, Y 61.3004, Z -6.3333, A 0.000, B 0.000, C 0.000 }
gfCNCPoint4[19611] = {X 493.7951, Y 63.2309, Z -6.3333, A 0.000, B 0.000, C 0.000 }
gfCNCPoint4[19612] = {X 493.2617, Y 65.1170, Z -6.3333, A 0.000, B 0.000, C 0.000 }
gfCNCPoint4[19613] = {X 492.5396, Y 66.9391, Z -6.3333, A 0.000, B 0.000, C 0.000 }
gfCNCPoint4[19614] = {X 491.6362, Y 68.6786, Z -6.3333, A 0.000, B 0.000, C 0.000 }
gfCNCPoint4[19615] = {X 490.5608, Y 70.3173, Z -6.3333, A 0.000, B 0.000, C 0.000 }
gfCNCPoint4[19616] = {X 490.5610, Y 83.2951, Z -6.3333, A 0.000, B 0.000, C 0.000 }
gfCNCPoint4[19617] = {X 507.6813, Y 83.2951, Z -6.3333, A 0.000, B 0.000, C 0.000 }
gfCNCPoint4[19618] = {X 507.6813, Y 85.6951, Z -6.3333, A 0.000, B 0.000, C 0.000 }
gfCNCPoint4[19619] = {X 585.6966, Y 85.6951, Z -6.3333, A 0.000, B 0.000, C 0.000 }
gfCNCPoint4[19620] = {X 585.6966, Y 63.3150, Z -6.3333, A 0.000, B 0.000, C 0.000 }
gfCNCPoint4[19621] = {X 584.3996, Y 63.5678, Z -6.3333, A 0.000, B 0.000, C 0.000 }
gfCNCPoint4[19622] = {X 583.0880, Y 63.7288, Z -6.3333, A 0.000, B 0.000, C 0.000 }
gfCNCPoint4[19623] = {X 581.1243, Y 63.7971, Z -6.3333, A 0.000, B 0.000, C 0.000 }
gfCNCPoint4[19624] = {X 579.1642, Y 63.6600, Z -6.3333, A 0.000, B 0.000, C 0.000 }
gfCNCPoint4[19625] = {X 577.2291, Y 63.3192, Z -6.3333, A 0.000, B 0.000, C 0.000 }
gfCNCPoint4[19626] = {X 575.3401, Y 62.7781, Z -6.3333, A 0.000, B 0.000, C 0.000 }
gfCNCPoint4[19627] = {X 573.3441, Y 63.3435, Z -6.3333, A 0.000, B 0.000, C 0.000 }
gfCNCPoint4[19628] = {X 571.2979, Y 63.6855, Z -6.3333, A 0.000, B 0.000, C 0.000 }
gfCNCPoint4[19629] = {X 569.2264, Y 63.8000, Z -6.3333, A 0.000, B 0.000, C 0.000 }
gfCNCPoint4[19630] = {X 562.4443, Y 63.8000, Z -6.3333, A 0.000, B 0.000, C 0.000 }
gfCNCPoint4[19631] = {X 560.5266, Y 63.7019, Z -6.3333, A 0.000, B 0.000, C 0.000 }
gfCNCPoint4[19632] = {X 558.6288, Y 63.4088, Z -6.3333, A 0.000, B 0.000, C 0.000 }
gfCNCPoint4[19633] = {X 556.7709, Y 62.9235, Z -6.3333, A 0.000, B 0.000, C 0.000 }
gfCNCPoint4[19634] = {X 554.9722, Y 62.2513, Z -6.3333, A 0.000, B 0.000, C 0.000 }
gfCNCPoint4[19635] = {X 553.2514, Y 61.3991, Z -6.3333, A 0.000, B 0.000, C 0.000 }
gfCNCPoint4[19636] = {X 551.6265, Y 60.3758, Z -6.3333, A 0.000, B 0.000, C 0.000 }
gfCNCPoint4[19637] = {X 550.1145, Y 59.1921, Z -6.3333, A 0.000, B 0.000, C 0.000 }
gfCNCPoint4[19638] = {X 548.7754, Y 57.9074, Z -6.3333, A 0.000, B 0.000, C 0.000 }
gfCNCPoint4[19639] = {X 547.5695, Y 56.4970, Z -6.3333, A 0.000, B 0.000, C 0.000 }
gfCNCPoint4[19640] = {X 546.2939, Y 56.8320, Z -6.3333, A 0.000, B 0.000, C 0.000 }
gfCNCPoint4[19641] = {X 544.9893, Y 57.0260, Z -6.3333, A 0.000, B 0.000, C 0.000 }
gfCNCPoint4[19642] = {X 543.6713, Y 57.0766, Z -6.3333, A 0.000, B 0.000, C 0.000 }
gfCNCPoint4[19643] = {X 526.9186, Y 57.0769, Z -6.3333, A 0.000, B 0.000, C 0.000 }
gfCNCPoint4[19644] = {X 525.4333, Y 57.8752, Z -6.3333, A 0.000, B 0.000, C 0.000 }
gfCNCPoint4[19645] = {X 523.8523, Y 58.4617, Z -6.3333, A 0.000, B 0.000, C 0.000 }
gfCNCPoint4[19646] = {X 522.2056, Y 58.8253, Z -6.3333, A 0.000, B 0.000, C 0.000 }
gfCNCPoint4[19647] = {X 520.5246, Y 58.9590, Z -6.3333, A 0.000, B 0.000, C 0.000 }
gfCNCPoint4[19648] = {X 519.7998, Y 58.9591, Z -6.3333, A 0.000, B 0.000, C 0.000 }
gfCNCPoint4[19649] = {X 518.2467, Y 58.8589, Z -6.3333, A 0.000, B 0.000, C 0.000 }
gfCNCPoint4[19650] = {X 516.7195, Y 58.5598, Z -6.3333, A 0.000, B 0.000, C 0.000 }
gfCNCPoint4[19651] = {X 515.2433, Y 58.0668, Z -6.3333, A 0.000, B 0.000, C 0.000 }
gfCNCPoint4[19652] = {X 513.8428, Y 57.3882, Z -6.3333, A 0.000, B 0.000, C 0.000 }
gfCNCPoint4[19653] = {X 512.5411, Y 56.5351, Z -6.3333, A 0.000, B 0.000, C 0.000 }
gfCNCPoint4[19654] = {X 511.3600, Y 55.5218, Z -6.3333, A 0.000, B 0.000, C 0.000 }
gfCNCPoint4[19655] = {X 510.3189, Y 54.3650, Z -6.3333, A 0.000, B 0.000, C 0.000 }
gfCNCPoint4[19656] = {X 508.9711, Y 55.3177, Z -6.3333, A 0.000, B 0.000, C 0.000 }
gfCNCPoint4[19657] = {X 507.5060, Y 56.0778, Z -6.3333, A 0.000, B 0.000, C 0.000 }
gfCNCPoint4[19658] = {X 505.9510, Y 56.6311, Z -6.3333, A 0.000, B 0.000, C 0.000 }
gfCNCPoint4[19659] = {X 504.3351, Y 56.9672, Z -6.3333, A 0.000, B 0.000, C 0.000 }
gfCNCPoint4[19660] = {X 502.6885, Y 57.0800, Z -6.3333, A 0.000, B 0.000, C 0.000 }
gfCNCPoint4[19661] = {X 496.2450, Y 57.0800, Z -6.3333, A 0.000, B 0.000, C 0.000 }
gfCNCPoint4[19662] = {X 495.4216, Y 57.0519, Z -6.3333, A 0.000, B 0.000, C 0.000 }
gfCNCPoint4[19663] = {X 494.6020, Y 56.9677, Z -6.3333, A 0.000, B 0.000, C 0.000 }
gfCNCPoint4[19664] = {X 493.1719, Y 56.6826, Z -6.3333, A 0.000, B 0.000, C 0.000 }
gfCNCPoint4[19665] = {X 491.7866, Y 56.2272, Z -6.3333, A 0.000, B 0.000, C 0.000 }
gfCNCPoint4[19666] = {X 491.8566, Y 57.1124, Z -6.3333, A 0.000, B 0.000, C 0.000 }
gfCNCPoint4[19667] = {X 491.8800, Y 58.0000, Z -6.3333, A 0.000, B 0.000, C 0.000 }
gfCNCPoint4[19668] = {X 491.8794, Y 59.0735, Z -6.3333, A 0.000, B 0.000, C 0.000 }
gfCNCPoint4[19669] = {X 491.8782, Y 59.1839, Z -6.3333, A 0.000, B 0.000, C 0.000 }
gfCNCPoint4[19670] = {X 491.8762, Y 59.2942, Z -6.3333, A 0.000, B 0.000, C 0.000 }
gfCNCPoint4[19671] = {X 491.7363, Y 61.1316, Z -6.3333, A 0.000, B 0.000, C 0.000 }
gfCNCPoint4[19672] = {X 491.3971, Y 62.9429, Z -6.3333, A 0.000, B 0.000, C 0.000 }
gfCNCPoint4[19673] = {X 490.8624, Y 64.7063, Z -6.3333, A 0.000, B 0.000, C 0.000 }
gfCNCPoint4[19674] = {X 490.1387, Y 66.4009, Z -6.3333, A 0.000, B 0.000, C 0.000 }
gfCNCPoint4[19675] = {X 489.2346, Y 68.0066, Z -6.3333, A 0.000, B 0.000, C 0.000 }
gfCNCPoint4[19676] = {X 488.1608, Y 69.5042, Z -6.3333, A 0.000, B 0.000, C 0.000 }
gfCNCPoint4[19677] = {X 488.1611, Y 85.6951, Z -6.3333, A 0.000, B 0.000, C 0.000 }
gfCNCPoint4[19678] = {X 507.6813, Y 85.6951, Z -6.3333, A 0.000, B 0.000, C 0.000 }
gfCNCPoint4[19679] = {X 507.6813, Y 88.0951, Z -6.3333, A 0.000, B 0.000, C 0.000 }
gfCNCPoint4[19680] = {X 588.0966, Y 88.0951, Z -6.3333, A 0.000, B 0.000, C 0.000 }
gfCNCPoint4[19681] = {X 588.0966, Y 60.4645, Z -6.3333, A 0.000, B 0.000, C 0.000 }
gfCNCPoint4[19682] = {X 587.7999, Y 60.3565, Z -6.3333, A 0.000, B 0.000, C 0.000 }
gfCNCPoint4[19683] = {X 587.5052, Y 60.2427, Z -6.3333, A 0.000, B 0.000, C 0.000 }
gfCNCPoint4[19684] = {X 586.3439, Y 60.6540, Z -6.3333, A 0.000, B 0.000, C 0.000 }
gfCNCPoint4[19685] = {X 585.1550, Y 60.9769, Z -6.3333, A 0.000, B 0.000, C 0.000 }
gfCNCPoint4[19686] = {X 583.5153, Y 61.2699, Z -6.3333, A 0.000, B 0.000, C 0.000 }
gfCNCPoint4[19687] = {X 581.8544, Y 61.3951, Z -6.3333, A 0.000, B 0.000, C 0.000 }
gfCNCPoint4[19688] = {X 580.1893, Y 61.3512, Z -6.3333, A 0.000, B 0.000, C 0.000 }
gfCNCPoint4[19689] = {X 578.5372, Y 61.1386, Z -6.3333, A 0.000, B 0.000, C 0.000 }
gfCNCPoint4[19690] = {X 576.9153, Y 60.7595, Z -6.3333, A 0.000, B 0.000, C 0.000 }
gfCNCPoint4[19691] = {X 575.3401, Y 60.2178, Z -6.3333, A 0.000, B 0.000, C 0.000 }
gfCNCPoint4[19692] = {X 573.8611, Y 60.7315, Z -6.3333, A 0.000, B 0.000, C 0.000 }
gfCNCPoint4[19693] = {X 572.3399, Y 61.1017, Z -6.3333, A 0.000, B 0.000, C 0.000 }
gfCNCPoint4[19694] = {X 570.7903, Y 61.3253, Z -6.3333, A 0.000, B 0.000, C 0.000 }
gfCNCPoint4[19695] = {X 569.2264, Y 61.4000, Z -6.3333, A 0.000, B 0.000, C 0.000 }
gfCNCPoint4[19696] = {X 562.4443, Y 61.4000, Z -6.3333, A 0.000, B 0.000, C 0.000 }
gfCNCPoint4[19697] = {X 560.4938, Y 61.2836, Z -6.3333, A 0.000, B 0.000, C 0.000 }
gfCNCPoint4[19698] = {X 558.5710, Y 60.9360, Z -6.3333, A 0.000, B 0.000, C 0.000 }
gfCNCPoint4[19699] = {X 556.7031, Y 60.3623, Z -6.3333, A 0.000, B 0.000, C 0.000 }
gfCNCPoint4[19700] = {X 554.9168, Y 59.5704, Z -6.3333, A 0.000, B 0.000, C 0.000 }
gfCNCPoint4[19701] = {X 553.2373, Y 58.5717, Z -6.3333, A 0.000, B 0.000, C 0.000 }
gfCNCPoint4[19702] = {X 551.6885, Y 57.3804, Z -6.3333, A 0.000, B 0.000, C 0.000 }
gfCNCPoint4[19703] = {X 550.4749, Y 56.2113, Z -6.3333, A 0.000, B 0.000, C 0.000 }
gfCNCPoint4[19704] = {X 549.3876, Y 54.9238, Z -6.3333, A 0.000, B 0.000, C 0.000 }
gfCNCPoint4[19705] = {X 548.4381, Y 53.5315, Z -6.3333, A 0.000, B 0.000, C 0.000 }
gfCNCPoint4[19706] = {X 547.3162, Y 54.0431, Z -6.3333, A 0.000, B 0.000, C 0.000 }
gfCNCPoint4[19707] = {X 546.1383, Y 54.4081, Z -6.3333, A 0.000, B 0.000, C 0.000 }
gfCNCPoint4[19708] = {X 544.9236, Y 54.6204, Z -6.3333, A 0.000, B 0.000, C 0.000 }
gfCNCPoint4[19709] = {X 543.6918, Y 54.6766, Z -6.3333, A 0.000, B 0.000, C 0.000 }
gfCNCPoint4[19710] = {X 526.1844, Y 54.6769, Z -6.3333, A 0.000, B 0.000, C 0.000 }
gfCNCPoint4[19711] = {X 524.8901, Y 55.4735, Z -6.3333, A 0.000, B 0.000, C 0.000 }
gfCNCPoint4[19712] = {X 523.4886, Y 56.0612, Z -6.3333, A 0.000, B 0.000, C 0.000 }
gfCNCPoint4[19713] = {X 522.0132, Y 56.4260, Z -6.3333, A 0.000, B 0.000, C 0.000 }
gfCNCPoint4[19714] = {X 520.4993, Y 56.5591, Z -6.3333, A 0.000, B 0.000, C 0.000 }
gfCNCPoint4[19715] = {X 519.7998, Y 56.5591, Z -6.3333, A 0.000, B 0.000, C 0.000 }
gfCNCPoint4[19716] = {X 518.3493, Y 56.4498, Z -6.3333, A 0.000, B 0.000, C 0.000 }
gfCNCPoint4[19717] = {X 516.9316, Y 56.1244, Z -6.3333, A 0.000, B 0.000, C 0.000 }
gfCNCPoint4[19718] = {X 515.5787, Y 55.5903, Z -6.3333, A 0.000, B 0.000, C 0.000 }
gfCNCPoint4[19719] = {X 514.3210, Y 54.8595, Z -6.3333, A 0.000, B 0.000, C 0.000 }
gfCNCPoint4[19720] = {X 513.1871, Y 53.9484, Z -6.3333, A 0.000, B 0.000, C 0.000 }
gfCNCPoint4[19721] = {X 512.2025, Y 52.8778, Z -6.3333, A 0.000, B 0.000, C 0.000 }
gfCNCPoint4[19722] = {X 511.3855, Y 51.6648, Z -6.3333, A 0.000, B 0.000, C 0.000 }
gfCNCPoint4[19723] = {X 510.7606, Y 50.3426, Z -6.3333, A 0.000, B 0.000, C 0.000 }
gfCNCPoint4[19724] = {X 509.8636, Y 51.4977, Z -6.3333, A 0.000, B 0.000, C 0.000 }
gfCNCPoint4[19725] = {X 508.8029, Y 52.5044, Z -6.3333, A 0.000, B 0.000, C 0.000 }
gfCNCPoint4[19726] = {X 507.7229, Y 53.2678, Z -6.3333, A 0.000, B 0.000, C 0.000 }
gfCNCPoint4[19727] = {X 506.5489, Y 53.8769, Z -6.3333, A 0.000, B 0.000, C 0.000 }
gfCNCPoint4[19728] = {X 505.3028, Y 54.3203, Z -6.3333, A 0.000, B 0.000, C 0.000 }
gfCNCPoint4[19729] = {X 504.0080, Y 54.5896, Z -6.3333, A 0.000, B 0.000, C 0.000 }
gfCNCPoint4[19730] = {X 502.6885, Y 54.6800, Z -6.3333, A 0.000, B 0.000, C 0.000 }
gfCNCPoint4[19731] = {X 496.2450, Y 54.6800, Z -6.3333, A 0.000, B 0.000, C 0.000 }
gfCNCPoint4[19732] = {X 495.0285, Y 54.6033, Z -6.3333, A 0.000, B 0.000, C 0.000 }
gfCNCPoint4[19733] = {X 493.8313, Y 54.3742, Z -6.3333, A 0.000, B 0.000, C 0.000 }
gfCNCPoint4[19734] = {X 492.6724, Y 53.9966, Z -6.3333, A 0.000, B 0.000, C 0.000 }
gfCNCPoint4[19735] = {X 491.4451, Y 53.4062, Z -6.3333, A 0.000, B 0.000, C 0.000 }
gfCNCPoint4[19736] = {X 490.3129, Y 52.6493, Z -6.3333, A 0.000, B 0.000, C 0.000 }
gfCNCPoint4[19737] = {X 489.2980, Y 51.7410, Z -6.3333, A 0.000, B 0.000, C 0.000 }
gfCNCPoint4[19738] = {X 488.8683, Y 52.1573, Z -6.3333, A 0.000, B 0.000, C 0.000 }
gfCNCPoint4[19739] = {X 488.4137, Y 52.5463, Z -6.3333, A 0.000, B 0.000, C 0.000 }
gfCNCPoint4[19740] = {X 488.8649, Y 53.8245, Z -6.3333, A 0.000, B 0.000, C 0.000 }
gfCNCPoint4[19741] = {X 489.1946, Y 55.1393, Z -6.3333, A 0.000, B 0.000, C 0.000 }
gfCNCPoint4[19742] = {X 489.3999, Y 56.4792, Z -6.3333, A 0.000, B 0.000, C 0.000 }
gfCNCPoint4[19743] = {X 489.4600, Y 57.2386, Z -6.3333, A 0.000, B 0.000, C 0.000 }
gfCNCPoint4[19744] = {X 489.4800, Y 58.0000, Z -6.3333, A 0.000, B 0.000, C 0.000 }
gfCNCPoint4[19745] = {X 489.4795, Y 59.0537, Z -6.3333, A 0.000, B 0.000, C 0.000 }
gfCNCPoint4[19746] = {X 489.3596, Y 60.7976, Z -6.3333, A 0.000, B 0.000, C 0.000 }
gfCNCPoint4[19747] = {X 489.0304, Y 62.5144, Z -6.3333, A 0.000, B 0.000, C 0.000 }
gfCNCPoint4[19748] = {X 488.4967, Y 64.1790, Z -6.3333, A 0.000, B 0.000, C 0.000 }
gfCNCPoint4[19749] = {X 487.7663, Y 65.7671, Z -6.3333, A 0.000, B 0.000, C 0.000 }
gfCNCPoint4[19750] = {X 486.8499, Y 67.2557, Z -6.3333, A 0.000, B 0.000, C 0.000 }
gfCNCPoint4[19751] = {X 485.7608, Y 68.6230, Z -6.3333, A 0.000, B 0.000, C 0.000 }
gfCNCPoint4[19752] = {X 485.7611, Y 87.3813, Z -6.3333, A 0.000, B 0.000, C 0.000 }
gfCNCPoint4[19753] = {X 486.0683, Y 87.7333, Z -6.3333, A 0.000, B 0.000, C 0.000 }
gfCNCPoint4[19754] = {X 486.3639, Y 88.0951, Z -6.3333, A 0.000, B 0.000, C 0.000 }
gfCNCPoint4[19755] = {X 507.6813, Y 88.0951, Z -6.3333, A 0.000, B 0.000, C 0.000 }
gfCNCPoint4[19756] = {X 507.6813, Y 90.4951, Z -6.3333, A 0.000, B 0.000, C 0.000 }
gfCNCPoint4[19757] = {X 590.4966, Y 90.4951, Z -6.3333, A 0.000, B 0.000, C 0.000 }
gfCNCPoint4[19758] = {X 590.4966, Y 58.6615, Z -6.3333, A 0.000, B 0.000, C 0.000 }
gfCNCPoint4[19759] = {X 588.9715, Y 58.2279, Z -6.3333, A 0.000, B 0.000, C 0.000 }
gfCNCPoint4[19760] = {X 587.5052, Y 57.6246, Z -6.3333, A 0.000, B 0.000, C 0.000 }
gfCNCPoint4[19761] = {X 585.8387, Y 58.2956, Z -6.3333, A 0.000, B 0.000, C 0.000 }
gfCNCPoint4[19762] = {X 584.0999, Y 58.7477, Z -6.3333, A 0.000, B 0.000, C 0.000 }
gfCNCPoint4[19763] = {X 582.3176, Y 58.9733, Z -6.3333, A 0.000, B 0.000, C 0.000 }
gfCNCPoint4[19764] = {X 580.5210, Y 58.9689, Z -6.3333, A 0.000, B 0.000, C 0.000 }
gfCNCPoint4[19765] = {X 578.7398, Y 58.7344, Z -6.3333, A 0.000, B 0.000, C 0.000 }
gfCNCPoint4[19766] = {X 577.0034, Y 58.2738, Z -6.3333, A 0.000, B 0.000, C 0.000 }
gfCNCPoint4[19767] = {X 575.3401, Y 57.5945, Z -6.3333, A 0.000, B 0.000, C 0.000 }
gfCNCPoint4[19768] = {X 573.8813, Y 58.2035, Z -6.3333, A 0.000, B 0.000, C 0.000 }
gfCNCPoint4[19769] = {X 572.3630, Y 58.6441, Z -6.3333, A 0.000, B 0.000, C 0.000 }
gfCNCPoint4[19770] = {X 570.8048, Y 58.9107, Z -6.3333, A 0.000, B 0.000, C 0.000 }
gfCNCPoint4[19771] = {X 569.2264, Y 59.0000, Z -6.3333, A 0.000, B 0.000, C 0.000 }
gfCNCPoint4[19772] = {X 562.4443, Y 59.0000, Z -6.3333, A 0.000, B 0.000, C 0.000 }
gfCNCPoint4[19773] = {X 560.7792, Y 58.9006, Z -6.3333, A 0.000, B 0.000, C 0.000 }
gfCNCPoint4[19774] = {X 559.1378, Y 58.6039, Z -6.3333, A 0.000, B 0.000, C 0.000 }
gfCNCPoint4[19775] = {X 557.5433, Y 58.1141, Z -6.3333, A 0.000, B 0.000, C 0.000 }
gfCNCPoint4[19776] = {X 556.0184, Y 57.4382, Z -6.3333, A 0.000, B 0.000, C 0.000 }
gfCNCPoint4[19777] = {X 554.5847, Y 56.5856, Z -6.3333, A 0.000, B 0.000, C 0.000 }
gfCNCPoint4[19778] = {X 553.2626, Y 55.5686, Z -6.3333, A 0.000, B 0.000, C 0.000 }
gfCNCPoint4[19779] = {X 552.2265, Y 54.5706, Z -6.3333, A 0.000, B 0.000, C 0.000 }
gfCNCPoint4[19780] = {X 551.2983, Y 53.4715, Z -6.3333, A 0.000, B 0.000, C 0.000 }
gfCNCPoint4[19781] = {X 550.4878, Y 52.2830, Z -6.3333, A 0.000, B 0.000, C 0.000 }
gfCNCPoint4[19782] = {X 549.8380, Y 51.0894, Z -6.3333, A 0.000, B 0.000, C 0.000 }
gfCNCPoint4[19783] = {X 549.3069, Y 49.8383, Z -6.3333, A 0.000, B 0.000, C 0.000 }
gfCNCPoint4[19784] = {X 548.3756, Y 50.7152, Z -6.3333, A 0.000, B 0.000, C 0.000 }
gfCNCPoint4[19785] = {X 547.3053, Y 51.4157, Z -6.3333, A 0.000, B 0.000, C 0.000 }
gfCNCPoint4[19786] = {X 546.1637, Y 51.9067, Z -6.3333, A 0.000, B 0.000, C 0.000 }
gfCNCPoint4[19787] = {X 544.9552, Y 52.1964, Z -6.3333, A 0.000, B 0.000, C 0.000 }
gfCNCPoint4[19788] = {X 543.7151, Y 52.2766, Z -6.3333, A 0.000, B 0.000, C 0.000 }
gfCNCPoint4[19789] = {X 525.3424, Y 52.2769, Z -6.3333, A 0.000, B 0.000, C 0.000 }
gfCNCPoint4[19790] = {X 524.2751, Y 53.0684, Z -6.3333, A 0.000, B 0.000, C 0.000 }
gfCNCPoint4[19791] = {X 523.0839, Y 53.6573, Z -6.3333, A 0.000, B 0.000, C 0.000 }
gfCNCPoint4[19792] = {X 521.8070, Y 54.0248, Z -6.3333, A 0.000, B 0.000, C 0.000 }
gfCNCPoint4[19793] = {X 520.4851, Y 54.1591, Z -6.3333, A 0.000, B 0.000, C 0.000 }
gfCNCPoint4[19794] = {X 519.7998, Y 54.1591, Z -6.3333, A 0.000, B 0.000, C 0.000 }
gfCNCPoint4[19795] = {X 518.5529, Y 54.0515, Z -6.3333, A 0.000, B 0.000, C 0.000 }
gfCNCPoint4[19796] = {X 517.3428, Y 53.7320, Z -6.3333, A 0.000, B 0.000, C 0.000 }
gfCNCPoint4[19797] = {X 516.2054, Y 53.2099, Z -6.3333, A 0.000, B 0.000, C 0.000 }
gfCNCPoint4[19798] = {X 515.1742, Y 52.5007, Z -6.3333, A 0.000, B 0.000, C 0.000 }
gfCNCPoint4[19799] = {X 514.2797, Y 51.6254, Z -6.3333, A 0.000, B 0.000, C 0.000 }
gfCNCPoint4[19800] = {X 513.5483, Y 50.6098, Z -6.3333, A 0.000, B 0.000, C 0.000 }
gfCNCPoint4[19801] = {X 513.0017, Y 49.4839, Z -6.3333, A 0.000, B 0.000, C 0.000 }
gfCNCPoint4[19802] = {X 512.7353, Y 48.6374, Z -6.3333, A 0.000, B 0.000, C 0.000 }
gfCNCPoint4[19803] = {X 512.5739, Y 47.7649, Z -6.3333, A 0.000, B 0.000, C 0.000 }
gfCNCPoint4[19804] = {X 512.5198, Y 46.8791, Z -6.3333, A 0.000, B 0.000, C 0.000 }
gfCNCPoint4[19805] = {X 512.5198, Y 39.9011, Z -6.3333, A 0.000, B 0.000, C 0.000 }
gfCNCPoint4[19806] = {X 512.5808, Y 38.9606, Z -6.3333, A 0.000, B 0.000, C 0.000 }
gfCNCPoint4[19807] = {X 512.7628, Y 38.0358, Z -6.3333, A 0.000, B 0.000, C 0.000 }
gfCNCPoint4[19808] = {X 513.0628, Y 37.1423, Z -6.3333, A 0.000, B 0.000, C 0.000 }
gfCNCPoint4[19809] = {X 513.5584, Y 36.1536, Z -6.3333, A 0.000, B 0.000, C 0.000 }
gfCNCPoint4[19810] = {X 514.1981, Y 35.2514, Z -6.3333, A 0.000, B 0.000, C 0.000 }
gfCNCPoint4[19811] = {X 514.9671, Y 34.4565, Z -6.3333, A 0.000, B 0.000, C 0.000 }
gfCNCPoint4[19812] = {X 515.8476, Y 33.7873, Z -6.3333, A 0.000, B 0.000, C 0.000 }
gfCNCPoint4[19813] = {X 513.2418, Y 29.7562, Z -6.3333, A 0.000, B 0.000, C 0.000 }
gfCNCPoint4[19814] = {X 513.5221, Y 29.5804, Z -6.3333, A 0.000, B 0.000, C 0.000 }
gfCNCPoint4[19815] = {X 513.8071, Y 29.4123, Z -6.3333, A 0.000, B 0.000, C 0.000 }
gfCNCPoint4[19816] = {X 513.8074, Y 27.6761, Z -6.3333, A 0.000, B 0.000, C 0.000 }
gfCNCPoint4[19817] = {X 513.5221, Y 27.5015, Z -6.3333, A 0.000, B 0.000, C 0.000 }
gfCNCPoint4[19818] = {X 513.2418, Y 27.3191, Z -6.3333, A 0.000, B 0.000, C 0.000 }
gfCNCPoint4[19819] = {X 513.2418, Y 29.7562, Z -6.3333, A 0.000, B 0.000, C 0.000 }
gfCNCPoint4[19820] = {X 514.5447, Y 31.7717, Z -6.3333, A 0.000, B 0.000, C 0.000 }
gfCNCPoint4[19821] = {X 515.3550, Y 31.3019, Z -6.3333, A 0.000, B 0.000, C 0.000 }
gfCNCPoint4[19822] = {X 516.2069, Y 30.9126, Z -6.3333, A 0.000, B 0.000, C 0.000 }
gfCNCPoint4[19823] = {X 516.2077, Y 26.2050, Z -6.3333, A 0.000, B 0.000, C 0.000 }
gfCNCPoint4[19824] = {X 515.3719, Y 25.8044, Z -6.3333, A 0.000, B 0.000, C 0.000 }
gfCNCPoint4[19825] = {X 514.5783, Y 25.3257, Z -6.3333, A 0.000, B 0.000, C 0.000 }
gfCNCPoint4[19826] = {X 513.5952, Y 24.5711, Z -6.3333, A 0.000, B 0.000, C 0.000 }
gfCNCPoint4[19827] = {X 512.7166, Y 23.6970, Z -6.3333, A 0.000, B 0.000, C 0.000 }
gfCNCPoint4[19828] = {X 511.9569, Y 22.7178, Z -6.3333, A 0.000, B 0.000, C 0.000 }
gfCNCPoint4[19829] = {X 511.3285, Y 21.6495, Z -6.3333, A 0.000, B 0.000, C 0.000 }
gfCNCPoint4[19830] = {X 510.8418, Y 20.5098, Z -6.3333, A 0.000, B 0.000, C 0.000 }
gfCNCPoint4[19831] = {X 510.8418, Y 36.2328, Z -6.3333, A 0.000, B 0.000, C 0.000 }
gfCNCPoint4[19832] = {X 511.5008, Y 34.9182, Z -6.3333, A 0.000, B 0.000, C 0.000 }
gfCNCPoint4[19833] = {X 512.3514, Y 33.7185, Z -6.3333, A 0.000, B 0.000, C 0.000 }
gfCNCPoint4[19834] = {X 513.3739, Y 32.6616, Z -6.3333, A 0.000, B 0.000, C 0.000 }
gfCNCPoint4[19835] = {X 514.5447, Y 31.7717, Z -6.3333, A 0.000, B 0.000, C 0.000 }
gfCNCPoint4[19836] = {X 515.8476, Y 33.7873, Z -6.3333, A 0.000, B 0.000, C 0.000 }
gfCNCPoint4[19837] = {X 516.7440, Y 33.2935, Z -6.3333, A 0.000, B 0.000, C 0.000 }
gfCNCPoint4[19838] = {X 517.7008, Y 32.9303, Z -6.3333, A 0.000, B 0.000, C 0.000 }
gfCNCPoint4[19839] = {X 518.6990, Y 32.7048, Z -6.3333, A 0.000, B 0.000, C 0.000 }
gfCNCPoint4[19840] = {X 518.6299, Y 32.1290, Z -6.3333, A 0.000, B 0.000, C 0.000 }
gfCNCPoint4[19841] = {X 518.6068, Y 31.5495, Z -6.3333, A 0.000, B 0.000, C 0.000 }
gfCNCPoint4[19842] = {X 518.6080, Y 24.4373, Z -6.3333, A 0.000, B 0.000, C 0.000 }
gfCNCPoint4[19843] = {X 517.3914, Y 24.0941, Z -6.3333, A 0.000, B 0.000, C 0.000 }
gfCNCPoint4[19844] = {X 516.2525, Y 23.5455, Z -6.3333, A 0.000, B 0.000, C 0.000 }
gfCNCPoint4[19845] = {X 515.2256, Y 22.8082, Z -6.3333, A 0.000, B 0.000, C 0.000 }
gfCNCPoint4[19846] = {X 514.3418, Y 21.9044, Z -6.3333, A 0.000, B 0.000, C 0.000 }
gfCNCPoint4[19847] = {X 513.6277, Y 20.8613, Z -6.3333, A 0.000, B 0.000, C 0.000 }
gfCNCPoint4[19848] = {X 513.1048, Y 19.7104, Z -6.3333, A 0.000, B 0.000, C 0.000 }
gfCNCPoint4[19849] = {X 512.7938, Y 18.5158, Z -6.3333, A 0.000, B 0.000, C 0.000 }
gfCNCPoint4[19850] = {X 512.6891, Y 17.2857, Z -6.3333, A 0.000, B 0.000, C 0.000 }
gfCNCPoint4[19851] = {X 512.6891, Y 10.3077, Z -6.3333, A 0.000, B 0.000, C 0.000 }
gfCNCPoint4[19852] = {X 512.7002, Y 9.9057, Z -6.3333, A 0.000, B 0.000, C 0.000 }
gfCNCPoint4[19853] = {X 512.7335, Y 9.5049, Z -6.3333, A 0.000, B 0.000, C 0.000 }
gfCNCPoint4[19854] = {X 509.4592, Y 9.5049, Z -6.3333, A 0.000, B 0.000, C 0.000 }
gfCNCPoint4[19855] = {X 509.7407, Y 10.3717, Z -6.3333, A 0.000, B 0.000, C 0.000 }
gfCNCPoint4[19856] = {X 509.9113, Y 11.2670, Z -6.3333, A 0.000, B 0.000, C 0.000 }
gfCNCPoint4[19857] = {X 509.9685, Y 12.1765, Z -6.3333, A 0.000, B 0.000, C 0.000 }
gfCNCPoint4[19858] = {X 509.9682, Y 13.0462, Z -6.3333, A 0.000, B 0.000, C 0.000 }
gfCNCPoint4[19859] = {X 509.8612, Y 14.2233, Z -6.3333, A 0.000, B 0.000, C 0.000 }
gfCNCPoint4[19860] = {X 509.5651, Y 15.3676, Z -6.3333, A 0.000, B 0.000, C 0.000 }
gfCNCPoint4[19861] = {X 509.0878, Y 16.4489, Z -6.3333, A 0.000, B 0.000, C 0.000 }
gfCNCPoint4[19862] = {X 508.4418, Y 17.4387, Z -6.3333, A 0.000, B 0.000, C 0.000 }
gfCNCPoint4[19863] = {X 508.4417, Y 39.7480, Z -6.3333, A 0.000, B 0.000, C 0.000 }
gfCNCPoint4[19864] = {X 509.0896, Y 40.7412, Z -6.3333, A 0.000, B 0.000, C 0.000 }
gfCNCPoint4[19865] = {X 509.5676, Y 41.8263, Z -6.3333, A 0.000, B 0.000, C 0.000 }
gfCNCPoint4[19866] = {X 509.8631, Y 42.9747, Z -6.3333, A 0.000, B 0.000, C 0.000 }
gfCNCPoint4[19867] = {X 509.9683, Y 44.1558, Z -6.3333, A 0.000, B 0.000, C 0.000 }
gfCNCPoint4[19868] = {X 509.9685, Y 45.0000, Z -6.3333, A 0.000, B 0.000, C 0.000 }
gfCNCPoint4[19869] = {X 509.8909, Y 46.0603, Z -6.3333, A 0.000, B 0.000, C 0.000 }
gfCNCPoint4[19870] = {X 509.6596, Y 47.0980, Z -6.3333, A 0.000, B 0.000, C 0.000 }
gfCNCPoint4[19871] = {X 509.2797, Y 48.0910, Z -6.3333, A 0.000, B 0.000, C 0.000 }
gfCNCPoint4[19872] = {X 508.7593, Y 49.0180, Z -6.3333, A 0.000, B 0.000, C 0.000 }
gfCNCPoint4[19873] = {X 508.0200, Y 49.9571, Z -6.3333, A 0.000, B 0.000, C 0.000 }
gfCNCPoint4[19874] = {X 507.1371, Y 50.7626, Z -6.3333, A 0.000, B 0.000, C 0.000 }
gfCNCPoint4[19875] = {X 506.1343, Y 51.4129, Z -6.3333, A 0.000, B 0.000, C 0.000 }
gfCNCPoint4[19876] = {X 505.0386, Y 51.8902, Z -6.3333, A 0.000, B 0.000, C 0.000 }
gfCNCPoint4[19877] = {X 503.8796, Y 52.1819, Z -6.3333, A 0.000, B 0.000, C 0.000 }
gfCNCPoint4[19878] = {X 502.6885, Y 52.2800, Z -6.3333, A 0.000, B 0.000, C 0.000 }
gfCNCPoint4[19879] = {X 496.2450, Y 52.2800, Z -6.3333, A 0.000, B 0.000, C 0.000 }
gfCNCPoint4[19880] = {X 495.0845, Y 52.1869, Z -6.3333, A 0.000, B 0.000, C 0.000 }
gfCNCPoint4[19881] = {X 493.9538, Y 51.9100, Z -6.3333, A 0.000, B 0.000, C 0.000 }
gfCNCPoint4[19882] = {X 492.8816, Y 51.4564, Z -6.3333, A 0.000, B 0.000, C 0.000 }
gfCNCPoint4[19883] = {X 491.8954, Y 50.8377, Z -6.3333, A 0.000, B 0.000, C 0.000 }
gfCNCPoint4[19884] = {X 491.0204, Y 50.0697, Z -6.3333, A 0.000, B 0.000, C 0.000 }
gfCNCPoint4[19885] = {X 490.2980, Y 49.1989, Z -6.3333, A 0.000, B 0.000, C 0.000 }
gfCNCPoint4[19886] = {X 489.7192, Y 48.2267, Z -6.3333, A 0.000, B 0.000, C 0.000 }
gfCNCPoint4[19887] = {X 489.2980, Y 47.1766, Z -6.3333, A 0.000, B 0.000, C 0.000 }
gfCNCPoint4[19888] = {X 488.8769, Y 48.2267, Z -6.3333, A 0.000, B 0.000, C 0.000 }
gfCNCPoint4[19889] = {X 488.2981, Y 49.1989, Z -6.3333, A 0.000, B 0.000, C 0.000 }
gfCNCPoint4[19890] = {X 487.5756, Y 50.0697, Z -6.3333, A 0.000, B 0.000, C 0.000 }
gfCNCPoint4[19891] = {X 486.8824, Y 50.6978, Z -6.3333, A 0.000, B 0.000, C 0.000 }
gfCNCPoint4[19892] = {X 486.1145, Y 51.2318, Z -6.3333, A 0.000, B 0.000, C 0.000 }
gfCNCPoint4[19893] = {X 485.2843, Y 51.6629, Z -6.3333, A 0.000, B 0.000, C 0.000 }
gfCNCPoint4[19894] = {X 486.0586, Y 53.1385, Z -6.3333, A 0.000, B 0.000, C 0.000 }
gfCNCPoint4[19895] = {X 486.6224, Y 54.7067, Z -6.3333, A 0.000, B 0.000, C 0.000 }
gfCNCPoint4[19896] = {X 486.9651, Y 56.3375, Z -6.3333, A 0.000, B 0.000, C 0.000 }
gfCNCPoint4[19897] = {X 487.0800, Y 58.0000, Z -6.3333, A 0.000, B 0.000, C 0.000 }
gfCNCPoint4[19898] = {X 487.0796, Y 59.0339, Z -6.3333, A 0.000, B 0.000, C 0.000 }
gfCNCPoint4[19899] = {X 486.9596, Y 60.6351, Z -6.3333, A 0.000, B 0.000, C 0.000 }
gfCNCPoint4[19900] = {X 486.6284, Y 62.2062, Z -6.3333, A 0.000, B 0.000, C 0.000 }
gfCNCPoint4[19901] = {X 486.0917, Y 63.7195, Z -6.3333, A 0.000, B 0.000, C 0.000 }
gfCNCPoint4[19902] = {X 485.3590, Y 65.1483, Z -6.3333, A 0.000, B 0.000, C 0.000 }
gfCNCPoint4[19903] = {X 484.4433, Y 66.4673, Z -6.3333, A 0.000, B 0.000, C 0.000 }
gfCNCPoint4[19904] = {X 483.3608, Y 67.6532, Z -6.3333, A 0.000, B 0.000, C 0.000 }
gfCNCPoint4[19905] = {X 483.3611, Y 88.3519, Z -6.3333, A 0.000, B 0.000, C 0.000 }
gfCNCPoint4[19906] = {X 484.3102, Y 89.3722, Z -6.3333, A 0.000, B 0.000, C 0.000 }
gfCNCPoint4[19907] = {X 485.1353, Y 90.4951, Z -6.3333, A 0.000, B 0.000, C 0.000 }
gfCNCPoint4[19908] = {X 507.6813, Y 90.4951, Z -6.3333, A 0.000, B 0.000, C 0.000 }
gfCNCPoint4[19909] = {X 507.6813, Y 92.8951, Z -6.3333, A 0.000, B 0.000, C 0.000 }
gfCNCPoint4[19910] = {X 592.8966, Y 92.8951, Z -6.3333, A 0.000, B 0.000, C 0.000 }
gfCNCPoint4[19911] = {X 592.8966, Y 56.5812, Z -6.3333, A 0.000, B 0.000, C 0.000 }
gfCNCPoint4[19912] = {X 591.4810, Y 56.4128, Z -6.3333, A 0.000, B 0.000, C 0.000 }
gfCNCPoint4[19913] = {X 590.0968, Y 56.0720, Z -6.3333, A 0.000, B 0.000, C 0.000 }
gfCNCPoint4[19914] = {X 588.7648, Y 55.5641, Z -6.3333, A 0.000, B 0.000, C 0.000 }
gfCNCPoint4[19915] = {X 587.5052, Y 54.8965, Z -6.3333, A 0.000, B 0.000, C 0.000 }
gfCNCPoint4[19916] = {X 586.9690, Y 55.2051, Z -6.3333, A 0.000, B 0.000, C 0.000 }
gfCNCPoint4[19917] = {X 586.4171, Y 55.4846, Z -6.3333, A 0.000, B 0.000, C 0.000 }
gfCNCPoint4[19918] = {X 584.8782, Y 56.0830, Z -6.3333, A 0.000, B 0.000, C 0.000 }
gfCNCPoint4[19919] = {X 583.2699, Y 56.4570, Z -6.3333, A 0.000, B 0.000, C 0.000 }
gfCNCPoint4[19920] = {X 581.6248, Y 56.5987, Z -6.3333, A 0.000, B 0.000, C 0.000 }
gfCNCPoint4[19921] = {X 579.9763, Y 56.5055, Z -6.3333, A 0.000, B 0.000, C 0.000 }
gfCNCPoint4[19922] = {X 578.3577, Y 56.1792, Z -6.3333, A 0.000, B 0.000, C 0.000 }
gfCNCPoint4[19923] = {X 576.8018, Y 55.6263, Z -6.3333, A 0.000, B 0.000, C 0.000 }
gfCNCPoint4[19924] = {X 575.3401, Y 54.8581, Z -6.3333, A 0.000, B 0.000, C 0.000 }
gfCNCPoint4[19925] = {X 573.9176, Y 55.6091, Z -6.3333, A 0.000, B 0.000, C 0.000 }
gfCNCPoint4[19926] = {X 572.4049, Y 56.1560, Z -6.3333, A 0.000, B 0.000, C 0.000 }
gfCNCPoint4[19927] = {X 570.8311, Y 56.4885, Z -6.3333, A 0.000, B 0.000, C 0.000 }
gfCNCPoint4[19928] = {X 569.2264, Y 56.6000, Z -6.3333, A 0.000, B 0.000, C 0.000 }
gfCNCPoint4[19929] = {X 562.4443, Y 56.6000, Z -6.3333, A 0.000, B 0.000, C 0.000 }
gfCNCPoint4[19930] = {X 560.7905, Y 56.4815, Z -6.3333, A 0.000, B 0.000, C 0.000 }
gfCNCPoint4[19931] = {X 559.1704, Y 56.1284, Z -6.3333, A 0.000, B 0.000, C 0.000 }
gfCNCPoint4[19932] = {X 557.6173, Y 55.5480, Z -6.3333, A 0.000, B 0.000, C 0.000 }
gfCNCPoint4[19933] = {X 556.1628, Y 54.7520, Z -6.3333, A 0.000, B 0.000, C 0.000 }
gfCNCPoint4[19934] = {X 554.8366, Y 53.7568, Z -6.3333, A 0.000, B 0.000, C 0.000 }
gfCNCPoint4[19935] = {X 553.7991, Y 52.7344, Z -6.3333, A 0.000, B 0.000, C 0.000 }
gfCNCPoint4[19936] = {X 552.8979, Y 51.5899, Z -6.3333, A 0.000, B 0.000, C 0.000 }
gfCNCPoint4[19937] = {X 552.1473, Y 50.3415, Z -6.3333, A 0.000, B 0.000, C 0.000 }
gfCNCPoint4[19938] = {X 551.5591, Y 49.0089, Z -6.3333, A 0.000, B 0.000, C 0.000 }
gfCNCPoint4[19939] = {X 551.1638, Y 47.7038, Z -6.3333, A 0.000, B 0.000, C 0.000 }
gfCNCPoint4[19940] = {X 550.9245, Y 46.3613, Z -6.3333, A 0.000, B 0.000, C 0.000 }
gfCNCPoint4[19941] = {X 550.8443, Y 45.0000, Z -6.3333, A 0.000, B 0.000, C 0.000 }
gfCNCPoint4[19942] = {X 550.8444, Y 44.0385, Z -6.3333, A 0.000, B 0.000, C 0.000 }
gfCNCPoint4[19943] = {X 550.9583, Y 42.4561, Z -6.3333, A 0.000, B 0.000, C 0.000 }
gfCNCPoint4[19944] = {X 551.2865, Y 40.9039, Z -6.3333, A 0.000, B 0.000, C 0.000 }
gfCNCPoint4[19945] = {X 551.8228, Y 39.4109, Z -6.3333, A 0.000, B 0.000, C 0.000 }
gfCNCPoint4[19946] = {X 549.6248, Y 38.4473, Z -6.3333, A 0.000, B 0.000, C 0.000 }
gfCNCPoint4[19947] = {X 549.7927, Y 38.0788, Z -6.3333, A 0.000, B 0.000, C 0.000 }
gfCNCPoint4[19948] = {X 549.9712, Y 37.7153, Z -6.3333, A 0.000, B 0.000, C 0.000 }
gfCNCPoint4[19949] = {X 549.9712, Y 16.9519, Z -6.3333, A 0.000, B 0.000, C 0.000 }
gfCNCPoint4[19950] = {X 549.8034, Y 17.1982, Z -6.3333, A 0.000, B 0.000, C 0.000 }
gfCNCPoint4[19951] = {X 549.6257, Y 17.4374, Z -6.3333, A 0.000, B 0.000, C 0.000 }
gfCNCPoint4[19952] = {X 549.6248, Y 38.4473, Z -6.3333, A 0.000, B 0.000, C 0.000 }
gfCNCPoint4[19953] = {X 551.8228, Y 39.4109, Z -6.3333, A 0.000, B 0.000, C 0.000 }
gfCNCPoint4[19954] = {X 552.0827, Y 38.8581, Z -6.3333, A 0.000, B 0.000, C 0.000 }
gfCNCPoint4[19955] = {X 552.3712, Y 38.3197, Z -6.3333, A 0.000, B 0.000, C 0.000 }
gfCNCPoint4[19956] = {X 552.3712, Y 11.6866, Z -6.3333, A 0.000, B 0.000, C 0.000 }
gfCNCPoint4[19957] = {X 551.6702, Y 10.2327, Z -6.3333, A 0.000, B 0.000, C 0.000 }
gfCNCPoint4[19958] = {X 551.1778, Y 8.6955, Z -6.3333, A 0.000, B 0.000, C 0.000 }
gfCNCPoint4[19959] = {X 550.9035, Y 7.1049, Z -6.3333, A 0.000, B 0.000, C 0.000 }
gfCNCPoint4[19960] = {X 524.2927, Y 7.1049, Z -6.3333, A 0.000, B 0.000, C 0.000 }
gfCNCPoint4[19961] = {X 524.3783, Y 7.2061, Z -6.3333, A 0.000, B 0.000, C 0.000 }
gfCNCPoint4[19962] = {X 524.4612, Y 7.3095, Z -6.3333, A 0.000, B 0.000, C 0.000 }
gfCNCPoint4[19963] = {X 543.7426, Y 7.3099, Z -6.3333, A 0.000, B 0.000, C 0.000 }
gfCNCPoint4[19964] = {X 544.7120, Y 7.3820, Z -6.3333, A 0.000, B 0.000, C 0.000 }
gfCNCPoint4[19965] = {X 545.6479, Y 7.6447, Z -6.3333, A 0.000, B 0.000, C 0.000 }
gfCNCPoint4[19966] = {X 546.5133, Y 8.0874, Z -6.3333, A 0.000, B 0.000, C 0.000 }
gfCNCPoint4[19967] = {X 547.2738, Y 8.6928, Z -6.3333, A 0.000, B 0.000, C 0.000 }
gfCNCPoint4[19968] = {X 547.8995, Y 9.4368, Z -6.3333, A 0.000, B 0.000, C 0.000 }
gfCNCPoint4[19969] = {X 548.3654, Y 10.2899, Z -6.3333, A 0.000, B 0.000, C 0.000 }
gfCNCPoint4[19970] = {X 548.6532, Y 11.2184, Z -6.3333, A 0.000, B 0.000, C 0.000 }
gfCNCPoint4[19971] = {X 548.7514, Y 12.1855, Z -6.3333, A 0.000, B 0.000, C 0.000 }
gfCNCPoint4[19972] = {X 548.7512, Y 13.0237, Z -6.3333, A 0.000, B 0.000, C 0.000 }
gfCNCPoint4[19973] = {X 548.6554, Y 13.9414, Z -6.3333, A 0.000, B 0.000, C 0.000 }
gfCNCPoint4[19974] = {X 548.3886, Y 14.8246, Z -6.3333, A 0.000, B 0.000, C 0.000 }
gfCNCPoint4[19975] = {X 547.9603, Y 15.6418, Z -6.3333, A 0.000, B 0.000, C 0.000 }
gfCNCPoint4[19976] = {X 547.6190, Y 16.1038, Z -6.3333, A 0.000, B 0.000, C 0.000 }
gfCNCPoint4[19977] = {X 547.2258, Y 16.5224, Z -6.3333, A 0.000, B 0.000, C 0.000 }
gfCNCPoint4[19978] = {X 547.2247, Y 40.6634, Z -6.3333, A 0.000, B 0.000, C 0.000 }
gfCNCPoint4[19979] = {X 547.8657, Y 41.4052, Z -6.3333, A 0.000, B 0.000, C 0.000 }
gfCNCPoint4[19980] = {X 548.3455, Y 42.2603, Z -6.3333, A 0.000, B 0.000, C 0.000 }
gfCNCPoint4[19981] = {X 548.6448, Y 43.1940, Z -6.3333, A 0.000, B 0.000, C 0.000 }
gfCNCPoint4[19982] = {X 548.7513, Y 44.1687, Z -6.3333, A 0.000, B 0.000, C 0.000 }
gfCNCPoint4[19983] = {X 548.7514, Y 45.0006, Z -6.3333, A 0.000, B 0.000, C 0.000 }
gfCNCPoint4[19984] = {X 548.6699, Y 45.8824, Z -6.3333, A 0.000, B 0.000, C 0.000 }
gfCNCPoint4[19985] = {X 548.4306, Y 46.7349, Z -6.3333, A 0.000, B 0.000, C 0.000 }
gfCNCPoint4[19986] = {X 548.0412, Y 47.5302, Z -6.3333, A 0.000, B 0.000, C 0.000 }
gfCNCPoint4[19987] = {X 547.5146, Y 48.2422, Z -6.3333, A 0.000, B 0.000, C 0.000 }
gfCNCPoint4[19988] = {X 546.7290, Y 48.9519, Z -6.3333, A 0.000, B 0.000, C 0.000 }
gfCNCPoint4[19989] = {X 545.8089, Y 49.4756, Z -6.3333, A 0.000, B 0.000, C 0.000 }
gfCNCPoint4[19990] = {X 544.7976, Y 49.7887, Z -6.3333, A 0.000, B 0.000, C 0.000 }
gfCNCPoint4[19991] = {X 543.7426, Y 49.8766, Z -6.3333, A 0.000, B 0.000, C 0.000 }
gfCNCPoint4[19992] = {X 524.3238, Y 49.8770, Z -6.3333, A 0.000, B 0.000, C 0.000 }
gfCNCPoint4[19993] = {X 523.7109, Y 50.5158, Z -6.3333, A 0.000, B 0.000, C 0.000 }
gfCNCPoint4[19994] = {X 522.9956, Y 51.0375, Z -6.3333, A 0.000, B 0.000, C 0.000 }
gfCNCPoint4[19995] = {X 522.2001, Y 51.4258, Z -6.3333, A 0.000, B 0.000, C 0.000 }
gfCNCPoint4[19996] = {X 521.3488, Y 51.6689, Z -6.3333, A 0.000, B 0.000, C 0.000 }
gfCNCPoint4[19997] = {X 520.4681, Y 51.7591, Z -6.3333, A 0.000, B 0.000, C 0.000 }
gfCNCPoint4[19998] = {X 519.7998, Y 51.7591, Z -6.3333, A 0.000, B 0.000, C 0.000 }
gfCNCPoint4[19999] = {X 518.8477, Y 51.6654, Z -6.3333, A 0.000, B 0.000, C 0.000 }
gfCNCPoint4[20000] = {X 517.9323, Y 51.3877, Z -6.3333, A 0.000, B 0.000, C 0.000 }
gfCNCPoint4[20001] = {X 517.0886, Y 50.9367, Z -6.3333, A 0.000, B 0.000, C 0.000 }
gfCNCPoint4[20002] = {X 516.3491, Y 50.3298, Z -6.3333, A 0.000, B 0.000, C 0.000 }
gfCNCPoint4[20003] = {X 515.7422, Y 49.5903, Z -6.3333, A 0.000, B 0.000, C 0.000 }
gfCNCPoint4[20004] = {X 515.2912, Y 48.7466, Z -6.3333, A 0.000, B 0.000, C 0.000 }
gfCNCPoint4[20005] = {X 515.0135, Y 47.8312, Z -6.3333, A 0.000, B 0.000, C 0.000 }
gfCNCPoint4[20006] = {X 514.9198, Y 46.8791, Z -6.3333, A 0.000, B 0.000, C 0.000 }
gfCNCPoint4[20007] = {X 514.9198, Y 39.9011, Z -6.3333, A 0.000, B 0.000, C 0.000 }
gfCNCPoint4[20008] = {X 515.0197, Y 38.9186, Z -6.3333, A 0.000, B 0.000, C 0.000 }
gfCNCPoint4[20009] = {X 515.3154, Y 37.9764, Z -6.3333, A 0.000, B 0.000, C 0.000 }
gfCNCPoint4[20010] = {X 515.7947, Y 37.1129, Z -6.3333, A 0.000, B 0.000, C 0.000 }
gfCNCPoint4[20011] = {X 516.4381, Y 36.3637, Z -6.3333, A 0.000, B 0.000, C 0.000 }
gfCNCPoint4[20012] = {X 517.2191, Y 35.7593, Z -6.3333, A 0.000, B 0.000, C 0.000 }
gfCNCPoint4[20013] = {X 518.1058, Y 35.3245, Z -6.3333, A 0.000, B 0.000, C 0.000 }
gfCNCPoint4[20014] = {X 519.0619, Y 35.0772, Z -6.3333, A 0.000, B 0.000, C 0.000 }
gfCNCPoint4[20015] = {X 519.4084, Y 35.0368, Z -6.3333, A 0.000, B 0.000, C 0.000 }
gfCNCPoint4[20016] = {X 519.7568, Y 35.0213, Z -6.3333, A 0.000, B 0.000, C 0.000 }
gfCNCPoint4[20017] = {X 520.5345, Y 35.0216, Z -6.3333, A 0.000, B 0.000, C 0.000 }
gfCNCPoint4[20018] = {X 521.4083, Y 35.1125, Z -6.3333, A 0.000, B 0.000, C 0.000 }
gfCNCPoint4[20019] = {X 522.2516, Y 35.3587, Z -6.3333, A 0.000, B 0.000, C 0.000 }
gfCNCPoint4[20020] = {X 523.0371, Y 35.7520, Z -6.3333, A 0.000, B 0.000, C 0.000 }
gfCNCPoint4[20021] = {X 523.7394, Y 36.2799, Z -6.3333, A 0.000, B 0.000, C 0.000 }
gfCNCPoint4[20022] = {X 524.3357, Y 36.9250, Z -6.3333, A 0.000, B 0.000, C 0.000 }
gfCNCPoint4[20023] = {X 534.0719, Y 36.9254, Z -6.3333, A 0.000, B 0.000, C 0.000 }
gfCNCPoint4[20024] = {X 534.0719, Y 34.5259, Z -6.3333, A 0.000, B 0.000, C 0.000 }
gfCNCPoint4[20025] = {X 530.3958, Y 34.5257, Z -6.3333, A 0.000, B 0.000, C 0.000 }
gfCNCPoint4[20026] = {X 529.7959, Y 35.1741, Z -6.3333, A 0.000, B 0.000, C 0.000 }
gfCNCPoint4[20027] = {X 529.0889, Y 35.7038, Z -6.3333, A 0.000, B 0.000, C 0.000 }
gfCNCPoint4[20028] = {X 528.2981, Y 36.0973, Z -6.3333, A 0.000, B 0.000, C 0.000 }
gfCNCPoint4[20029] = {X 527.4493, Y 36.3418, Z -6.3333, A 0.000, B 0.000, C 0.000 }
gfCNCPoint4[20030] = {X 526.5703, Y 36.4293, Z -6.3333, A 0.000, B 0.000, C 0.000 }
gfCNCPoint4[20031] = {X 525.8868, Y 36.4294, Z -6.3333, A 0.000, B 0.000, C 0.000 }
gfCNCPoint4[20032] = {X 524.9094, Y 36.3306, Z -6.3333, A 0.000, B 0.000, C 0.000 }
gfCNCPoint4[20033] = {X 523.9717, Y 36.0380, Z -6.3333, A 0.000, B 0.000, C 0.000 }
gfCNCPoint4[20034] = {X 523.1116, Y 35.5636, Z -6.3333, A 0.000, B 0.000, C 0.000 }
gfCNCPoint4[20035] = {X 522.3639, Y 34.9265, Z -6.3333, A 0.000, B 0.000, C 0.000 }
gfCNCPoint4[20036] = {X 521.7590, Y 34.1525, Z -6.3333, A 0.000, B 0.000, C 0.000 }
gfCNCPoint4[20037] = {X 521.3213, Y 33.2731, Z -6.3333, A 0.000, B 0.000, C 0.000 }
gfCNCPoint4[20038] = {X 521.0686, Y 32.3239, Z -6.3333, A 0.000, B 0.000, C 0.000 }
gfCNCPoint4[20039] = {X 521.0222, Y 31.9379, Z -6.3333, A 0.000, B 0.000, C 0.000 }
gfCNCPoint4[20040] = {X 521.0068, Y 31.5495, Z -6.3333, A 0.000, B 0.000, C 0.000 }
gfCNCPoint4[20041] = {X 521.0076, Y 24.4815, Z -6.3333, A 0.000, B 0.000, C 0.000 }
gfCNCPoint4[20042] = {X 521.0984, Y 23.6300, Z -6.3333, A 0.000, B 0.000, C 0.000 }
gfCNCPoint4[20043] = {X 521.3368, Y 22.8074, Z -6.3333, A 0.000, B 0.000, C 0.000 }
gfCNCPoint4[20044] = {X 521.7152, Y 22.0391, Z -6.3333, A 0.000, B 0.000, C 0.000 }
gfCNCPoint4[20045] = {X 521.1864, Y 22.1316, Z -6.3333, A 0.000, B 0.000, C 0.000 }
gfCNCPoint4[20046] = {X 520.6505, Y 22.1656, Z -6.3333, A 0.000, B 0.000, C 0.000 }
gfCNCPoint4[20047] = {X 519.9691, Y 22.1657, Z -6.3333, A 0.000, B 0.000, C 0.000 }
gfCNCPoint4[20048] = {X 519.5109, Y 22.1442, Z -6.3333, A 0.000, B 0.000, C 0.000 }
gfCNCPoint4[20049] = {X 519.0567, Y 22.0797, Z -6.3333, A 0.000, B 0.000, C 0.000 }
gfCNCPoint4[20050] = {X 518.1336, Y 21.8074, Z -6.3333, A 0.000, B 0.000, C 0.000 }
gfCNCPoint4[20051] = {X 517.2820, Y 21.3592, Z -6.3333, A 0.000, B 0.000, C 0.000 }
gfCNCPoint4[20052] = {X 516.5348, Y 20.7527, Z -6.3333, A 0.000, B 0.000, C 0.000 }
gfCNCPoint4[20053] = {X 515.9212, Y 20.0113, Z -6.3333, A 0.000, B 0.000, C 0.000 }
gfCNCPoint4[20054] = {X 515.4650, Y 19.1639, Z -6.3333, A 0.000, B 0.000, C 0.000 }
gfCNCPoint4[20055] = {X 515.1840, Y 18.2434, Z -6.3333, A 0.000, B 0.000, C 0.000 }
gfCNCPoint4[20056] = {X 515.0891, Y 17.2857, Z -6.3333, A 0.000, B 0.000, C 0.000 }
gfCNCPoint4[20057] = {X 515.0891, Y 10.3077, Z -6.3333, A 0.000, B 0.000, C 0.000 }
gfCNCPoint4[20058] = {X 515.0966, Y 10.0382, Z -6.3333, A 0.000, B 0.000, C 0.000 }
gfCNCPoint4[20059] = {X 515.1189, Y 9.7696, Z -6.3333, A 0.000, B 0.000, C 0.000 }
gfCNCPoint4[20060] = {X 515.3252, Y 8.8083, Z -6.3333, A 0.000, B 0.000, C 0.000 }
gfCNCPoint4[20061] = {X 515.7199, Y 7.9079, Z -6.3333, A 0.000, B 0.000, C 0.000 }
gfCNCPoint4[20062] = {X 516.2872, Y 7.1049, Z -6.3333, A 0.000, B 0.000, C 0.000 }
gfCNCPoint4[20063] = {X 516.6493, Y 7.4199, Z -6.3333, A 0.000, B 0.000, C 0.000 }
gfCNCPoint4[20064] = {X 517.3374, Y 6.7815, Z -6.3333, A 0.000, B 0.000, C 0.000 }
gfCNCPoint4[20065] = {X 518.1452, Y 6.3035, Z -6.3333, A 0.000, B 0.000, C 0.000 }
gfCNCPoint4[20066] = {X 519.0360, Y 6.0078, Z -6.3333, A 0.000, B 0.000, C 0.000 }
gfCNCPoint4[20067] = {X 519.9692, Y 5.9077, Z -6.3333, A 0.000, B 0.000, C 0.000 }
gfCNCPoint4[20068] = {X 520.6509, Y 5.9079, Z -6.3333, A 0.000, B 0.000, C 0.000 }
gfCNCPoint4[20069] = {X 521.4832, Y 5.9950, Z -6.3333, A 0.000, B 0.000, C 0.000 }
gfCNCPoint4[20070] = {X 522.2839, Y 6.2382, Z -6.3333, A 0.000, B 0.000, C 0.000 }
gfCNCPoint4[20071] = {X 523.0240, Y 6.6285, Z -6.3333, A 0.000, B 0.000, C 0.000 }
gfCNCPoint4[20072] = {X 523.6769, Y 7.1520, Z -6.3333, A 0.000, B 0.000, C 0.000 }
gfCNCPoint4[20073] = {X 524.2189, Y 7.7895, Z -6.3333, A 0.000, B 0.000, C 0.000 }
gfCNCPoint4[20074] = {X 543.7489, Y 7.7899, Z -6.3333, A 0.000, B 0.000, C 0.000 }
gfCNCPoint4[20075] = {X 544.7472, Y 7.8772, Z -6.3333, A 0.000, B 0.000, C 0.000 }
gfCNCPoint4[20076] = {X 545.6999, Y 8.1879, Z -6.3333, A 0.000, B 0.000, C 0.000 }
gfCNCPoint4[20077] = {X 546.5577, Y 8.7059, Z -6.3333, A 0.000, B 0.000, C 0.000 }
gfCNCPoint4[20078] = {X 547.2763, Y 9.4044, Z -6.3333, A 0.000, B 0.000, C 0.000 }
gfCNCPoint4[20079] = {X 547.8183, Y 10.2473, Z -6.3333, A 0.000, B 0.000, C 0.000 }
gfCNCPoint4[20080] = {X 548.1559, Y 11.1908, Z -6.3333, A 0.000, B 0.000, C 0.000 }
gfCNCPoint4[20081] = {X 548.2714, Y 12.1862, Z -6.3333, A 0.000, B 0.000, C 0.000 }
gfCNCPoint4[20082] = {X 548.2712, Y 13.0233, Z -6.3333, A 0.000, B 0.000, C 0.000 }
gfCNCPoint4[20083] = {X 548.1630, Y 13.9487, Z -6.3333, A 0.000, B 0.000, C 0.000 }
gfCNCPoint4[20084] = {X 547.8624, Y 14.8306, Z -6.3333, A 0.000, B 0.000, C 0.000 }
gfCNCPoint4[20085] = {X 547.3828, Y 15.6295, Z -6.3333, A 0.000, B 0.000, C 0.000 }
gfCNCPoint4[20086] = {X 546.7458, Y 16.3094, Z -6.3333, A 0.000, B 0.000, C 0.000 }
gfCNCPoint4[20087] = {X 546.7447, Y 40.8764, Z -6.3333, A 0.000, B 0.000, C 0.000 }
gfCNCPoint4[20088] = {X 547.3890, Y 41.5655, Z -6.3333, A 0.000, B 0.000, C 0.000 }
gfCNCPoint4[20089] = {X 547.8716, Y 42.3761, Z -6.3333, A 0.000, B 0.000, C 0.000 }
gfCNCPoint4[20090] = {X 548.1703, Y 43.2709, Z -6.3333, A 0.000, B 0.000, C 0.000 }
gfCNCPoint4[20091] = {X 548.2714, Y 44.2089, Z -6.3333, A 0.000, B 0.000, C 0.000 }
gfCNCPoint4[20092] = {X 548.2714, Y 45.0006, Z -6.3333, A 0.000, B 0.000, C 0.000 }
gfCNCPoint4[20093] = {X 548.1559, Y 45.9960, Z -6.3333, A 0.000, B 0.000, C 0.000 }
gfCNCPoint4[20094] = {X 547.8183, Y 46.9395, Z -6.3333, A 0.000, B 0.000, C 0.000 }
gfCNCPoint4[20095] = {X 547.2762, Y 47.7823, Z -6.3333, A 0.000, B 0.000, C 0.000 }
gfCNCPoint4[20096] = {X 546.5577, Y 48.4808, Z -6.3333, A 0.000, B 0.000, C 0.000 }
gfCNCPoint4[20097] = {X 545.6998, Y 48.9987, Z -6.3333, A 0.000, B 0.000, C 0.000 }
gfCNCPoint4[20098] = {X 544.7471, Y 49.3093, Z -6.3333, A 0.000, B 0.000, C 0.000 }
gfCNCPoint4[20099] = {X 543.7489, Y 49.3966, Z -6.3333, A 0.000, B 0.000, C 0.000 }
gfCNCPoint4[20100] = {X 524.0865, Y 49.3970, Z -6.3333, A 0.000, B 0.000, C 0.000 }
gfCNCPoint4[20101] = {X 523.5297, Y 50.0319, Z -6.3333, A 0.000, B 0.000, C 0.000 }
gfCNCPoint4[20102] = {X 522.8652, Y 50.5532, Z -6.3333, A 0.000, B 0.000, C 0.000 }
gfCNCPoint4[20103] = {X 522.1160, Y 50.9430, Z -6.3333, A 0.000, B 0.000, C 0.000 }
gfCNCPoint4[20104] = {X 521.3077, Y 51.1877, Z -6.3333, A 0.000, B 0.000, C 0.000 }
gfCNCPoint4[20105] = {X 520.4681, Y 51.2791, Z -6.3333, A 0.000, B 0.000, C 0.000 }
gfCNCPoint4[20106] = {X 519.7998, Y 51.2791, Z -6.3333, A 0.000, B 0.000, C 0.000 }
gfCNCPoint4[20107] = {X 518.8207, Y 51.1688, Z -6.3333, A 0.000, B 0.000, C 0.000 }
gfCNCPoint4[20108] = {X 517.8907, Y 50.8434, Z -6.3333, A 0.000, B 0.000, C 0.000 }
gfCNCPoint4[20109] = {X 517.0564, Y 50.3192, Z -6.3333, A 0.000, B 0.000, C 0.000 }
gfCNCPoint4[20110] = {X 516.3597, Y 49.6225, Z -6.3333, A 0.000, B 0.000, C 0.000 }
gfCNCPoint4[20111] = {X 515.8355, Y 48.7882, Z -6.3333, A 0.000, B 0.000, C 0.000 }
gfCNCPoint4[20112] = {X 515.5101, Y 47.8582, Z -6.3333, A 0.000, B 0.000, C 0.000 }
gfCNCPoint4[20113] = {X 515.3998, Y 46.8791, Z -6.3333, A 0.000, B 0.000, C 0.000 }
gfCNCPoint4[20114] = {X 515.3998, Y 39.9011, Z -6.3333, A 0.000, B 0.000, C 0.000 }
gfCNCPoint4[20115] = {X 515.5101, Y 38.9220, Z -6.3333, A 0.000, B 0.000, C 0.000 }
gfCNCPoint4[20116] = {X 515.8355, Y 37.9920, Z -6.3333, A 0.000, B 0.000, C 0.000 }
gfCNCPoint4[20117] = {X 516.3597, Y 37.1577, Z -6.3333, A 0.000, B 0.000, C 0.000 }
gfCNCPoint4[20118] = {X 517.0564, Y 36.4610, Z -6.3333, A 0.000, B 0.000, C 0.000 }
gfCNCPoint4[20119] = {X 517.8907, Y 35.9368, Z -6.3333, A 0.000, B 0.000, C 0.000 }
gfCNCPoint4[20120] = {X 518.8207, Y 35.6114, Z -6.3333, A 0.000, B 0.000, C 0.000 }
gfCNCPoint4[20121] = {X 519.7998, Y 35.5011, Z -6.3333, A 0.000, B 0.000, C 0.000 }
gfCNCPoint4[20122] = {X 520.5280, Y 35.5015, Z -6.3333, A 0.000, B 0.000, C 0.000 }
gfCNCPoint4[20123] = {X 521.3612, Y 35.5927, Z -6.3333, A 0.000, B 0.000, C 0.000 }
gfCNCPoint4[20124] = {X 522.1621, Y 35.8402, Z -6.3333, A 0.000, B 0.000, C 0.000 }
gfCNCPoint4[20125] = {X 522.9015, Y 36.2352, Z -6.3333, A 0.000, B 0.000, C 0.000 }
gfCNCPoint4[20126] = {X 523.5525, Y 36.7631, Z -6.3333, A 0.000, B 0.000, C 0.000 }
gfCNCPoint4[20127] = {X 524.0917, Y 37.4050, Z -6.3333, A 0.000, B 0.000, C 0.000 }
gfCNCPoint4[20128] = {X 534.5519, Y 37.4054, Z -6.3333, A 0.000, B 0.000, C 0.000 }
gfCNCPoint4[20129] = {X 534.5519, Y 34.0460, Z -6.3333, A 0.000, B 0.000, C 0.000 }
gfCNCPoint4[20130] = {X 530.1518, Y 34.0457, Z -6.3333, A 0.000, B 0.000, C 0.000 }
gfCNCPoint4[20131] = {X 529.6041, Y 34.6959, Z -6.3333, A 0.000, B 0.000, C 0.000 }
gfCNCPoint4[20132] = {X 528.9416, Y 35.2286, Z -6.3333, A 0.000, B 0.000, C 0.000 }
gfCNCPoint4[20133] = {X 528.1890, Y 35.6241, Z -6.3333, A 0.000, B 0.000, C 0.000 }
gfCNCPoint4[20134] = {X 527.3745, Y 35.8673, Z -6.3333, A 0.000, B 0.000, C 0.000 }
gfCNCPoint4[20135] = {X 526.5283, Y 35.9495, Z -6.3333, A 0.000, B 0.000, C 0.000 }
gfCNCPoint4[20136] = {X 525.8868, Y 35.9495, Z -6.3333, A 0.000, B 0.000, C 0.000 }
gfCNCPoint4[20137] = {X 524.9077, Y 35.8391, Z -6.3333, A 0.000, B 0.000, C 0.000 }
gfCNCPoint4[20138] = {X 523.9777, Y 35.5137, Z -6.3333, A 0.000, B 0.000, C 0.000 }
gfCNCPoint4[20139] = {X 523.1434, Y 34.9895, Z -6.3333, A 0.000, B 0.000, C 0.000 }
gfCNCPoint4[20140] = {X 522.4467, Y 34.2928, Z -6.3333, A 0.000, B 0.000, C 0.000 }
gfCNCPoint4[20141] = {X 521.9225, Y 33.4585, Z -6.3333, A 0.000, B 0.000, C 0.000 }
gfCNCPoint4[20142] = {X 521.5971, Y 32.5285, Z -6.3333, A 0.000, B 0.000, C 0.000 }
gfCNCPoint4[20143] = {X 521.4868, Y 31.5495, Z -6.3333, A 0.000, B 0.000, C 0.000 }
gfCNCPoint4[20144] = {X 521.4868, Y 24.5714, Z -6.3333, A 0.000, B 0.000, C 0.000 }
gfCNCPoint4[20145] = {X 521.5971, Y 23.5923, Z -6.3333, A 0.000, B 0.000, C 0.000 }
gfCNCPoint4[20146] = {X 521.9225, Y 22.6623, Z -6.3333, A 0.000, B 0.000, C 0.000 }
gfCNCPoint4[20147] = {X 522.4467, Y 21.8281, Z -6.3333, A 0.000, B 0.000, C 0.000 }
gfCNCPoint4[20148] = {X 523.1434, Y 21.1314, Z -6.3333, A 0.000, B 0.000, C 0.000 }
gfCNCPoint4[20149] = {X 523.9777, Y 20.6072, Z -6.3333, A 0.000, B 0.000, C 0.000 }
gfCNCPoint4[20150] = {X 524.9077, Y 20.2817, Z -6.3333, A 0.000, B 0.000, C 0.000 }
gfCNCPoint4[20151] = {X 525.8868, Y 20.1714, Z -6.3333, A 0.000, B 0.000, C 0.000 }
gfCNCPoint4[20152] = {X 526.5702, Y 20.1716, Z -6.3333, A 0.000, B 0.000, C 0.000 }
gfCNCPoint4[20153] = {X 527.2693, Y 20.2342, Z -6.3333, A 0.000, B 0.000, C 0.000 }
gfCNCPoint4[20154] = {X 527.9494, Y 20.4072, Z -6.3333, A 0.000, B 0.000, C 0.000 }
gfCNCPoint4[20155] = {X 528.5934, Y 20.6861, Z -6.3333, A 0.000, B 0.000, C 0.000 }
gfCNCPoint4[20156] = {X 528.8187, Y 20.2623, Z -6.3333, A 0.000, B 0.000, C 0.000 }
gfCNCPoint4[20157] = {X 534.0719, Y 20.2624, Z -6.3333, A 0.000, B 0.000, C 0.000 }
gfCNCPoint4[20158] = {X 534.0719, Y 21.5734, Z -6.3333, A 0.000, B 0.000, C 0.000 }
gfCNCPoint4[20159] = {X 530.3788, Y 21.5732, Z -6.3333, A 0.000, B 0.000, C 0.000 }
gfCNCPoint4[20160] = {X 529.6679, Y 20.8354, Z -6.3333, A 0.000, B 0.000, C 0.000 }
gfCNCPoint4[20161] = {X 528.8187, Y 20.2623, Z -6.3333, A 0.000, B 0.000, C 0.000 }
gfCNCPoint4[20162] = {X 528.5934, Y 20.6861, Z -6.3333, A 0.000, B 0.000, C 0.000 }
gfCNCPoint4[20163] = {X 529.1778, Y 21.0585, Z -6.3333, A 0.000, B 0.000, C 0.000 }
gfCNCPoint4[20164] = {X 529.6965, Y 21.5180, Z -6.3333, A 0.000, B 0.000, C 0.000 }
gfCNCPoint4[20165] = {X 530.1366, Y 22.0532, Z -6.3333, A 0.000, B 0.000, C 0.000 }
gfCNCPoint4[20166] = {X 534.5519, Y 22.0534, Z -6.3333, A 0.000, B 0.000, C 0.000 }
gfCNCPoint4[20167] = {X 534.5519, Y 19.7824, Z -6.3333, A 0.000, B 0.000, C 0.000 }
gfCNCPoint4[20168] = {X 524.2340, Y 19.7822, Z -6.3333, A 0.000, B 0.000, C 0.000 }
gfCNCPoint4[20169] = {X 523.6863, Y 20.4323, Z -6.3333, A 0.000, B 0.000, C 0.000 }
gfCNCPoint4[20170] = {X 523.0239, Y 20.9650, Z -6.3333, A 0.000, B 0.000, C 0.000 }
gfCNCPoint4[20171] = {X 522.2713, Y 21.3603, Z -6.3333, A 0.000, B 0.000, C 0.000 }
gfCNCPoint4[20172] = {X 521.4568, Y 21.6036, Z -6.3333, A 0.000, B 0.000, C 0.000 }
gfCNCPoint4[20173] = {X 520.6107, Y 21.6857, Z -6.3333, A 0.000, B 0.000, C 0.000 }
gfCNCPoint4[20174] = {X 519.9691, Y 21.6857, Z -6.3333, A 0.000, B 0.000, C 0.000 }
gfCNCPoint4[20175] = {X 518.9900, Y 21.5754, Z -6.3333, A 0.000, B 0.000, C 0.000 }
gfCNCPoint4[20176] = {X 518.0600, Y 21.2500, Z -6.3333, A 0.000, B 0.000, C 0.000 }
gfCNCPoint4[20177] = {X 517.2257, Y 20.7258, Z -6.3333, A 0.000, B 0.000, C 0.000 }
gfCNCPoint4[20178] = {X 516.5290, Y 20.0291, Z -6.3333, A 0.000, B 0.000, C 0.000 }
gfCNCPoint4[20179] = {X 516.0048, Y 19.1948, Z -6.3333, A 0.000, B 0.000, C 0.000 }
gfCNCPoint4[20180] = {X 515.6794, Y 18.2648, Z -6.3333, A 0.000, B 0.000, C 0.000 }
gfCNCPoint4[20181] = {X 515.5691, Y 17.2857, Z -6.3333, A 0.000, B 0.000, C 0.000 }
gfCNCPoint4[20182] = {X 515.5691, Y 10.3077, Z -6.3333, A 0.000, B 0.000, C 0.000 }
gfCNCPoint4[20183] = {X 515.6394, Y 9.5244, Z -6.3333, A 0.000, B 0.000, C 0.000 }
gfCNCPoint4[20184] = {X 515.8480, Y 8.7661, Z -6.3333, A 0.000, B 0.000, C 0.000 }
gfCNCPoint4[20185] = {X 516.1883, Y 8.0571, Z -6.3333, A 0.000, B 0.000, C 0.000 }
gfCNCPoint4[20186] = {X 516.6493, Y 7.4199, Z -6.3333, A 0.000, B 0.000, C 0.000 }
gfCNCPoint4[20187] = {X 516.2872, Y 7.1049, Z -6.3333, A 0.000, B 0.000, C 0.000 }
gfCNCPoint4[20188] = {X 469.2601, Y 7.1049, Z -6.3333, A 0.000, B 0.000, C 0.000 }
gfCNCPoint4[20189] = {X 469.2601, Y 11.9049, Z -6.3333, A 0.000, B 0.000, C 0.000 }
gfCNCPoint4[20190] = {X 469.1140, Y 11.9049, Z -6.3333, A 0.000, B 0.000, C 0.000 }
gfCNCPoint4[20191] = {X 469.1170, Y 12.0430, Z -6.3333, A 0.000, B 0.000, C 0.000 }
gfCNCPoint4[20192] = {X 469.1179, Y 12.1812, Z -6.3333, A 0.000, B 0.000, C 0.000 }
gfCNCPoint4[20193] = {X 469.1884, Y 12.0427, Z -6.3333, A 0.000, B 0.000, C 0.000 }
gfCNCPoint4[20194] = {X 469.2601, Y 11.9049, Z -6.3333, A 0.000, B 0.000, C 0.000 }
gfCNCPoint4[20195] = {X 469.2601, Y 9.5049, Z -6.3333, A 0.000, B 0.000, C 0.000 }
gfCNCPoint4[20196] = {X 466.2076, Y 9.5049, Z -6.3333, A 0.000, B 0.000, C 0.000 }
gfCNCPoint4[20197] = {X 466.5690, Y 10.7170, Z -6.3333, A 0.000, B 0.000, C 0.000 }
gfCNCPoint4[20198] = {X 466.7150, Y 11.9734, Z -6.3333, A 0.000, B 0.000, C 0.000 }
gfCNCPoint4[20199] = {X 466.7172, Y 12.0772, Z -6.3333, A 0.000, B 0.000, C 0.000 }
gfCNCPoint4[20200] = {X 466.7179, Y 12.1810, Z -6.3333, A 0.000, B 0.000, C 0.000 }
gfCNCPoint4[20201] = {X 466.7179, Y 12.9779, Z -6.3333, A 0.000, B 0.000, C 0.000 }
gfCNCPoint4[20202] = {X 466.6192, Y 14.1731, Z -6.3333, A 0.000, B 0.000, C 0.000 }
gfCNCPoint4[20203] = {X 466.3256, Y 15.3358, Z -6.3333, A 0.000, B 0.000, C 0.000 }
gfCNCPoint4[20204] = {X 465.8450, Y 16.4345, Z -6.3333, A 0.000, B 0.000, C 0.000 }
gfCNCPoint4[20205] = {X 465.1907, Y 17.4395, Z -6.3333, A 0.000, B 0.000, C 0.000 }
gfCNCPoint4[20206] = {X 465.1910, Y 25.8840, Z -6.3333, A 0.000, B 0.000, C 0.000 }
gfCNCPoint4[20207] = {X 467.5910, Y 25.8839, Z -6.3333, A 0.000, B 0.000, C 0.000 }
gfCNCPoint4[20208] = {X 467.5916, Y 38.9914, Z -6.3333, A 0.000, B 0.000, C 0.000 }
gfCNCPoint4[20209] = {X 467.6015, Y 39.0069, Z -6.3333, A 0.000, B 0.000, C 0.000 }
gfCNCPoint4[20210] = {X 468.3506, Y 37.9855, Z -6.3333, A 0.000, B 0.000, C 0.000 }
gfCNCPoint4[20211] = {X 469.2267, Y 37.0706, Z -6.3333, A 0.000, B 0.000, C 0.000 }
gfCNCPoint4[20212] = {X 470.2148, Y 36.2780, Z -6.3333, A 0.000, B 0.000, C 0.000 }
gfCNCPoint4[20213] = {X 471.5270, Y 33.7095, Z -6.3333, A 0.000, B 0.000, C 0.000 }
gfCNCPoint4[20214] = {X 470.4795, Y 32.4131, Z -6.3333, A 0.000, B 0.000, C 0.000 }
gfCNCPoint4[20215] = {X 469.5654, Y 31.0194, Z -6.3333, A 0.000, B 0.000, C 0.000 }
gfCNCPoint4[20216] = {X 468.7939, Y 29.5420, Z -6.3333, A 0.000, B 0.000, C 0.000 }
gfCNCPoint4[20217] = {X 468.1724, Y 27.9955, Z -6.3333, A 0.000, B 0.000, C 0.000 }
gfCNCPoint4[20218] = {X 467.7071, Y 26.3950, Z -6.3333, A 0.000, B 0.000, C 0.000 }
gfCNCPoint4[20219] = {X 467.6476, Y 26.1398, Z -6.3333, A 0.000, B 0.000, C 0.000 }
gfCNCPoint4[20220] = {X 467.5910, Y 25.8839, Z -6.3333, A 0.000, B 0.000, C 0.000 }
gfCNCPoint4[20221] = {X 465.1910, Y 25.8840, Z -6.3333, A 0.000, B 0.000, C 0.000 }
gfCNCPoint4[20222] = {X 465.1916, Y 39.7485, Z -6.3333, A 0.000, B 0.000, C 0.000 }
gfCNCPoint4[20223] = {X 465.3908, Y 40.0181, Z -6.3333, A 0.000, B 0.000, C 0.000 }
gfCNCPoint4[20224] = {X 465.5774, Y 40.2966, Z -6.3333, A 0.000, B 0.000, C 0.000 }
gfCNCPoint4[20225] = {X 466.0634, Y 41.1919, Z -6.3333, A 0.000, B 0.000, C 0.000 }
gfCNCPoint4[20226] = {X 466.4196, Y 42.1462, Z -6.3333, A 0.000, B 0.000, C 0.000 }
gfCNCPoint4[20227] = {X 466.6392, Y 43.1408, Z -6.3333, A 0.000, B 0.000, C 0.000 }
gfCNCPoint4[20228] = {X 466.7178, Y 44.1564, Z -6.3333, A 0.000, B 0.000, C 0.000 }
gfCNCPoint4[20229] = {X 466.7179, Y 45.0000, Z -6.3333, A 0.000, B 0.000, C 0.000 }
gfCNCPoint4[20230] = {X 466.7033, Y 45.4609, Z -6.3333, A 0.000, B 0.000, C 0.000 }
gfCNCPoint4[20231] = {X 466.6596, Y 45.9200, Z -6.3333, A 0.000, B 0.000, C 0.000 }
gfCNCPoint4[20232] = {X 468.5433, Y 45.9200, Z -6.3333, A 0.000, B 0.000, C 0.000 }
gfCNCPoint4[20233] = {X 468.4996, Y 45.4609, Z -6.3333, A 0.000, B 0.000, C 0.000 }
gfCNCPoint4[20234] = {X 468.4850, Y 45.0000, Z -6.3333, A 0.000, B 0.000, C 0.000 }
gfCNCPoint4[20235] = {X 468.4850, Y 44.2089, Z -6.3333, A 0.000, B 0.000, C 0.000 }
gfCNCPoint4[20236] = {X 468.5580, Y 43.1798, Z -6.3333, A 0.000, B 0.000, C 0.000 }
gfCNCPoint4[20237] = {X 468.7759, Y 42.1713, Z -6.3333, A 0.000, B 0.000, C 0.000 }
gfCNCPoint4[20238] = {X 469.1341, Y 41.2038, Z -6.3333, A 0.000, B 0.000, C 0.000 }
gfCNCPoint4[20239] = {X 469.6255, Y 40.2966, Z -6.3333, A 0.000, B 0.000, C 0.000 }
gfCNCPoint4[20240] = {X 470.3102, Y 39.3876, Z -6.3333, A 0.000, B 0.000, C 0.000 }
gfCNCPoint4[20241] = {X 471.1282, Y 38.5964, Z -6.3333, A 0.000, B 0.000, C 0.000 }
gfCNCPoint4[20242] = {X 472.0595, Y 37.9424, Z -6.3333, A 0.000, B 0.000, C 0.000 }
gfCNCPoint4[20243] = {X 474.4564, Y 33.2507, Z -6.3333, A 0.000, B 0.000, C 0.000 }
gfCNCPoint4[20244] = {X 473.2243, Y 32.0061, Z -6.3333, A 0.000, B 0.000, C 0.000 }
gfCNCPoint4[20245] = {X 472.1523, Y 30.6211, Z -6.3333, A 0.000, B 0.000, C 0.000 }
gfCNCPoint4[20246] = {X 471.2561, Y 29.1164, Z -6.3333, A 0.000, B 0.000, C 0.000 }
gfCNCPoint4[20247] = {X 470.5491, Y 27.5141, Z -6.3333, A 0.000, B 0.000, C 0.000 }
gfCNCPoint4[20248] = {X 470.0416, Y 25.8379, Z -6.3333, A 0.000, B 0.000, C 0.000 }
gfCNCPoint4[20249] = {X 469.9882, Y 25.6093, Z -6.3333, A 0.000, B 0.000, C 0.000 }
gfCNCPoint4[20250] = {X 469.9375, Y 25.3801, Z -6.3333, A 0.000, B 0.000, C 0.000 }
gfCNCPoint4[20251] = {X 469.6264, Y 23.4852, Z -6.3333, A 0.000, B 0.000, C 0.000 }
gfCNCPoint4[20252] = {X 469.5012, Y 21.5689, Z -6.3333, A 0.000, B 0.000, C 0.000 }
gfCNCPoint4[20253] = {X 469.5632, Y 19.6496, Z -6.3333, A 0.000, B 0.000, C 0.000 }
gfCNCPoint4[20254] = {X 469.8118, Y 17.7455, Z -6.3333, A 0.000, B 0.000, C 0.000 }
gfCNCPoint4[20255] = {X 470.2446, Y 15.8746, Z -6.3333, A 0.000, B 0.000, C 0.000 }
gfCNCPoint4[20256] = {X 470.6912, Y 14.5429, Z -6.3333, A 0.000, B 0.000, C 0.000 }
gfCNCPoint4[20257] = {X 471.2620, Y 13.2596, Z -6.3333, A 0.000, B 0.000, C 0.000 }
gfCNCPoint4[20258] = {X 471.3226, Y 13.1405, Z -6.3333, A 0.000, B 0.000, C 0.000 }
gfCNCPoint4[20259] = {X 471.3843, Y 13.0219, Z -6.3333, A 0.000, B 0.000, C 0.000 }
gfCNCPoint4[20260] = {X 472.1254, Y 11.7667, Z -6.3333, A 0.000, B 0.000, C 0.000 }
gfCNCPoint4[20261] = {X 472.9865, Y 10.5906, Z -6.3333, A 0.000, B 0.000, C 0.000 }
gfCNCPoint4[20262] = {X 473.9591, Y 9.5049, Z -6.3333, A 0.000, B 0.000, C 0.000 }
gfCNCPoint4[20263] = {X 469.2601, Y 9.5049, Z -6.3333, A 0.000, B 0.000, C 0.000 }
gfCNCPoint4[20264] = {X 469.2601, Y 7.1049, Z -6.3333, A 0.000, B 0.000, C 0.000 }
gfCNCPoint4[20265] = {X 370.0953, Y 7.1049, Z -6.3333, A 0.000, B 0.000, C 0.000 }
gfCNCPoint4[20266] = {X 371.1186, Y 8.7930, Z -6.3333, A 0.000, B 0.000, C 0.000 }
gfCNCPoint4[20267] = {X 372.0303, Y 10.5439, Z -6.3333, A 0.000, B 0.000, C 0.000 }
gfCNCPoint4[20268] = {X 372.8772, Y 12.4761, Z -6.3333, A 0.000, B 0.000, C 0.000 }
gfCNCPoint4[20269] = {X 373.5884, Y 14.4623, Z -6.3333, A 0.000, B 0.000, C 0.000 }
gfCNCPoint4[20270] = {X 374.1603, Y 16.4930, Z -6.3333, A 0.000, B 0.000, C 0.000 }
gfCNCPoint4[20271] = {X 374.5903, Y 18.5584, Z -6.3333, A 0.000, B 0.000, C 0.000 }
gfCNCPoint4[20272] = {X 374.9755, Y 21.3233, Z -6.3333, A 0.000, B 0.000, C 0.000 }
gfCNCPoint4[20273] = {X 375.1518, Y 24.1093, Z -6.3333, A 0.000, B 0.000, C 0.000 }
gfCNCPoint4[20274] = {X 375.1181, Y 26.9007, Z -6.3333, A 0.000, B 0.000, C 0.000 }
gfCNCPoint4[20275] = {X 374.8746, Y 29.6816, Z -6.3333, A 0.000, B 0.000, C 0.000 }
gfCNCPoint4[20276] = {X 374.4228, Y 32.4364, Z -6.3333, A 0.000, B 0.000, C 0.000 }
gfCNCPoint4[20277] = {X 373.7859, Y 34.9943, Z -6.3333, A 0.000, B 0.000, C 0.000 }
gfCNCPoint4[20278] = {X 372.9262, Y 37.4862, Z -6.3333, A 0.000, B 0.000, C 0.000 }
gfCNCPoint4[20279] = {X 371.8503, Y 39.8926, Z -6.3333, A 0.000, B 0.000, C 0.000 }
gfCNCPoint4[20280] = {X 370.5666, Y 42.1949, Z -6.3333, A 0.000, B 0.000, C 0.000 }
gfCNCPoint4[20281] = {X 369.0850, Y 44.3751, Z -6.3333, A 0.000, B 0.000, C 0.000 }
gfCNCPoint4[20282] = {X 368.9669, Y 44.5368, Z -6.3333, A 0.000, B 0.000, C 0.000 }
gfCNCPoint4[20283] = {X 367.5696, Y 46.2481, Z -6.3333, A 0.000, B 0.000, C 0.000 }
gfCNCPoint4[20284] = {X 366.0388, Y 47.8411, Z -6.3333, A 0.000, B 0.000, C 0.000 }
gfCNCPoint4[20285] = {X 364.3843, Y 49.3053, Z -6.3333, A 0.000, B 0.000, C 0.000 }
gfCNCPoint4[20286] = {X 362.6171, Y 50.6312, Z -6.3333, A 0.000, B 0.000, C 0.000 }
gfCNCPoint4[20287] = {X 360.7485, Y 51.8101, Z -6.3333, A 0.000, B 0.000, C 0.000 }
gfCNCPoint4[20288] = {X 358.7910, Y 52.8343, Z -6.3333, A 0.000, B 0.000, C 0.000 }
gfCNCPoint4[20289] = {X 358.6058, Y 52.9209, Z -6.3333, A 0.000, B 0.000, C 0.000 }
gfCNCPoint4[20290] = {X 358.4200, Y 53.0062, Z -6.3333, A 0.000, B 0.000, C 0.000 }
gfCNCPoint4[20291] = {X 356.1466, Y 53.8828, Z -6.3333, A 0.000, B 0.000, C 0.000 }
gfCNCPoint4[20292] = {X 353.8064, Y 54.5612, Z -6.3333, A 0.000, B 0.000, C 0.000 }
gfCNCPoint4[20293] = {X 351.4167, Y 55.0365, Z -6.3333, A 0.000, B 0.000, C 0.000 }
gfCNCPoint4[20294] = {X 348.9949, Y 55.3050, Z -6.3333, A 0.000, B 0.000, C 0.000 }
gfCNCPoint4[20295] = {X 349.9661, Y 69.6722, Z -6.3333, A 0.000, B 0.000, C 0.000 }
gfCNCPoint4[20296] = {X 348.6648, Y 69.7403, Z -6.3333, A 0.000, B 0.000, C 0.000 }
gfCNCPoint4[20297] = {X 347.3620, Y 69.7687, Z -6.3333, A 0.000, B 0.000, C 0.000 }
gfCNCPoint4[20298] = {X 346.5844, Y 69.7778, Z -6.3333, A 0.000, B 0.000, C 0.000 }
gfCNCPoint4[20299] = {X 345.8069, Y 69.7731, Z -6.3333, A 0.000, B 0.000, C 0.000 }
gfCNCPoint4[20300] = {X 345.5912, Y 70.1904, Z -6.3333, A 0.000, B 0.000, C 0.000 }
gfCNCPoint4[20301] = {X 345.3675, Y 70.6035, Z -6.3333, A 0.000, B 0.000, C 0.000 }
gfCNCPoint4[20302] = {X 347.2077, Y 70.6208, Z -6.3333, A 0.000, B 0.000, C 0.000 }
gfCNCPoint4[20303] = {X 349.0480, Y 70.6091, Z -6.3333, A 0.000, B 0.000, C 0.000 }
gfCNCPoint4[20304] = {X 349.7518, Y 70.6088, Z -6.3333, A 0.000, B 0.000, C 0.000 }
gfCNCPoint4[20305] = {X 350.4556, Y 70.6032, Z -6.3333, A 0.000, B 0.000, C 0.000 }
gfCNCPoint4[20306] = {X 350.2058, Y 70.1404, Z -6.3333, A 0.000, B 0.000, C 0.000 }
gfCNCPoint4[20307] = {X 349.9661, Y 69.6722, Z -6.3333, A 0.000, B 0.000, C 0.000 }
gfCNCPoint4[20308] = {X 349.8042, Y 67.2776, Z -6.3333, A 0.000, B 0.000, C 0.000 }
gfCNCPoint4[20309] = {X 348.5675, Y 67.3422, Z -6.3333, A 0.000, B 0.000, C 0.000 }
gfCNCPoint4[20310] = {X 347.3293, Y 67.3688, Z -6.3333, A 0.000, B 0.000, C 0.000 }
gfCNCPoint4[20311] = {X 345.8126, Y 67.3729, Z -6.3333, A 0.000, B 0.000, C 0.000 }
gfCNCPoint4[20312] = {X 344.2968, Y 67.3210, Z -6.3333, A 0.000, B 0.000, C 0.000 }
gfCNCPoint4[20313] = {X 343.8113, Y 68.3945, Z -6.3333, A 0.000, B 0.000, C 0.000 }
gfCNCPoint4[20314] = {X 343.2684, Y 69.4400, Z -6.3333, A 0.000, B 0.000, C 0.000 }
gfCNCPoint4[20315] = {X 342.7884, Y 70.2630, Z -6.3333, A 0.000, B 0.000, C 0.000 }
gfCNCPoint4[20316] = {X 342.2728, Y 71.0640, Z -6.3333, A 0.000, B 0.000, C 0.000 }
gfCNCPoint4[20317] = {X 342.2730, Y 72.9111, Z -6.3333, A 0.000, B 0.000, C 0.000 }
gfCNCPoint4[20318] = {X 343.7992, Y 72.9669, Z -6.3333, A 0.000, B 0.000, C 0.000 }
gfCNCPoint4[20319] = {X 345.3260, Y 73.0031, Z -6.3333, A 0.000, B 0.000, C 0.000 }
gfCNCPoint4[20320] = {X 347.1936, Y 73.0208, Z -6.3333, A 0.000, B 0.000, C 0.000 }
gfCNCPoint4[20321] = {X 349.0612, Y 73.0091, Z -6.3333, A 0.000, B 0.000, C 0.000 }
gfCNCPoint4[20322] = {X 349.7724, Y 73.0087, Z -6.3333, A 0.000, B 0.000, C 0.000 }
gfCNCPoint4[20323] = {X 350.4835, Y 73.0030, Z -6.3333, A 0.000, B 0.000, C 0.000 }
gfCNCPoint4[20324] = {X 352.0214, Y 72.9730, Z -6.3333, A 0.000, B 0.000, C 0.000 }
gfCNCPoint4[20325] = {X 353.5587, Y 72.9185, Z -6.3333, A 0.000, B 0.000, C 0.000 }
gfCNCPoint4[20326] = {X 353.5586, Y 71.0764, Z -6.3333, A 0.000, B 0.000, C 0.000 }
gfCNCPoint4[20327] = {X 353.0387, Y 70.2694, Z -6.3333, A 0.000, B 0.000, C 0.000 }
gfCNCPoint4[20328] = {X 352.5550, Y 69.4402, Z -6.3333, A 0.000, B 0.000, C 0.000 }
gfCNCPoint4[20329] = {X 351.9680, Y 68.3027, Z -6.3333, A 0.000, B 0.000, C 0.000 }
gfCNCPoint4[20330] = {X 351.4492, Y 67.1326, Z -6.3333, A 0.000, B 0.000, C 0.000 }
gfCNCPoint4[20331] = {X 350.6275, Y 67.2135, Z -6.3333, A 0.000, B 0.000, C 0.000 }
gfCNCPoint4[20332] = {X 349.8042, Y 67.2776, Z -6.3333, A 0.000, B 0.000, C 0.000 }
gfCNCPoint4[20333] = {X 349.6424, Y 64.8831, Z -6.3333, A 0.000, B 0.000, C 0.000 }
gfCNCPoint4[20334] = {X 348.4701, Y 64.9442, Z -6.3333, A 0.000, B 0.000, C 0.000 }
gfCNCPoint4[20335] = {X 347.2966, Y 64.9690, Z -6.3333, A 0.000, B 0.000, C 0.000 }
gfCNCPoint4[20336] = {X 344.9827, Y 64.9498, Z -6.3333, A 0.000, B 0.000, C 0.000 }
gfCNCPoint4[20337] = {X 342.6740, Y 64.7925, Z -6.3333, A 0.000, B 0.000, C 0.000 }
gfCNCPoint4[20338] = {X 341.9394, Y 66.7272, Z -6.3333, A 0.000, B 0.000, C 0.000 }
gfCNCPoint4[20339] = {X 341.0020, Y 68.5721, Z -6.3333, A 0.000, B 0.000, C 0.000 }
gfCNCPoint4[20340] = {X 339.8727, Y 70.3062, Z -6.3333, A 0.000, B 0.000, C 0.000 }
gfCNCPoint4[20341] = {X 339.8732, Y 75.1884, Z -6.3333, A 0.000, B 0.000, C 0.000 }
gfCNCPoint4[20342] = {X 344.4717, Y 75.3860, Z -6.3333, A 0.000, B 0.000, C 0.000 }
gfCNCPoint4[20343] = {X 349.0745, Y 75.4092, Z -6.3333, A 0.000, B 0.000, C 0.000 }
gfCNCPoint4[20344] = {X 352.5186, Y 75.3593, Z -6.3333, A 0.000, B 0.000, C 0.000 }
gfCNCPoint4[20345] = {X 355.9589, Y 75.1901, Z -6.3333, A 0.000, B 0.000, C 0.000 }
gfCNCPoint4[20346] = {X 355.9586, Y 70.3175, Z -6.3333, A 0.000, B 0.000, C 0.000 }
gfCNCPoint4[20347] = {X 355.0510, Y 68.9597, Z -6.3333, A 0.000, B 0.000, C 0.000 }
gfCNCPoint4[20348] = {X 354.2616, Y 67.5300, Z -6.3333, A 0.000, B 0.000, C 0.000 }
gfCNCPoint4[20349] = {X 353.5960, Y 66.0386, Z -6.3333, A 0.000, B 0.000, C 0.000 }
gfCNCPoint4[20350] = {X 353.0590, Y 64.4962, Z -6.3333, A 0.000, B 0.000, C 0.000 }
gfCNCPoint4[20351] = {X 351.3551, Y 64.7283, Z -6.3333, A 0.000, B 0.000, C 0.000 }
gfCNCPoint4[20352] = {X 349.6424, Y 64.8831, Z -6.3333, A 0.000, B 0.000, C 0.000 }
gfCNCPoint4[20353] = {X 349.4805, Y 62.4886, Z -6.3333, A 0.000, B 0.000, C 0.000 }
gfCNCPoint4[20354] = {X 348.3728, Y 62.5461, Z -6.3333, A 0.000, B 0.000, C 0.000 }
gfCNCPoint4[20355] = {X 347.2639, Y 62.5691, Z -6.3333, A 0.000, B 0.000, C 0.000 }
gfCNCPoint4[20356] = {X 345.1284, Y 62.5535, Z -6.3333, A 0.000, B 0.000, C 0.000 }
gfCNCPoint4[20357] = {X 342.9975, Y 62.4127, Z -6.3333, A 0.000, B 0.000, C 0.000 }
gfCNCPoint4[20358] = {X 340.8786, Y 62.1470, Z -6.3333, A 0.000, B 0.000, C 0.000 }
gfCNCPoint4[20359] = {X 340.4888, Y 63.7347, Z -6.3333, A 0.000, B 0.000, C 0.000 }
gfCNCPoint4[20360] = {X 339.9476, Y 65.2774, Z -6.3333, A 0.000, B 0.000, C 0.000 }
gfCNCPoint4[20361] = {X 339.2600, Y 66.7607, Z -6.3333, A 0.000, B 0.000, C 0.000 }
gfCNCPoint4[20362] = {X 338.4325, Y 68.1707, Z -6.3333, A 0.000, B 0.000, C 0.000 }
gfCNCPoint4[20363] = {X 337.4727, Y 69.4942, Z -6.3333, A 0.000, B 0.000, C 0.000 }
gfCNCPoint4[20364] = {X 337.4734, Y 77.4237, Z -6.3333, A 0.000, B 0.000, C 0.000 }
gfCNCPoint4[20365] = {X 341.3402, Y 77.6733, Z -6.3333, A 0.000, B 0.000, C 0.000 }
gfCNCPoint4[20366] = {X 345.2129, Y 77.8019, Z -6.3333, A 0.000, B 0.000, C 0.000 }
gfCNCPoint4[20367] = {X 349.0878, Y 77.8092, Z -6.3333, A 0.000, B 0.000, C 0.000 }
gfCNCPoint4[20368] = {X 353.7279, Y 77.7157, Z -6.3333, A 0.000, B 0.000, C 0.000 }
gfCNCPoint4[20369] = {X 358.3590, Y 77.4107, Z -6.3333, A 0.000, B 0.000, C 0.000 }
gfCNCPoint4[20370] = {X 358.3585, Y 69.5043, Z -6.3333, A 0.000, B 0.000, C 0.000 }
gfCNCPoint4[20371] = {X 357.3476, Y 68.1046, Z -6.3333, A 0.000, B 0.000, C 0.000 }
gfCNCPoint4[20372] = {X 356.4850, Y 66.6089, Z -6.3333, A 0.000, B 0.000, C 0.000 }
gfCNCPoint4[20373] = {X 355.7796, Y 65.0330, Z -6.3333, A 0.000, B 0.000, C 0.000 }
gfCNCPoint4[20374] = {X 355.2389, Y 63.3933, Z -6.3333, A 0.000, B 0.000, C 0.000 }
gfCNCPoint4[20375] = {X 354.8686, Y 61.7069, Z -6.3333, A 0.000, B 0.000, C 0.000 }
gfCNCPoint4[20376] = {X 352.1895, Y 62.2009, Z -6.3333, A 0.000, B 0.000, C 0.000 }
gfCNCPoint4[20377] = {X 349.4805, Y 62.4886, Z -6.3333, A 0.000, B 0.000, C 0.000 }
gfCNCPoint4[20378] = {X 349.3187, Y 60.0940, Z -6.3333, A 0.000, B 0.000, C 0.000 }
gfCNCPoint4[20379] = {X 348.2755, Y 60.1481, Z -6.3333, A 0.000, B 0.000, C 0.000 }
gfCNCPoint4[20380] = {X 347.2313, Y 60.1692, Z -6.3333, A 0.000, B 0.000, C 0.000 }
gfCNCPoint4[20381] = {X 344.3951, Y 60.1151, Z -6.3333, A 0.000, B 0.000, C 0.000 }
gfCNCPoint4[20382] = {X 341.5733, Y 59.8245, Z -6.3333, A 0.000, B 0.000, C 0.000 }
gfCNCPoint4[20383] = {X 338.7856, Y 59.2994, Z -6.3333, A 0.000, B 0.000, C 0.000 }
gfCNCPoint4[20384] = {X 338.6400, Y 60.9987, Z -6.3333, A 0.000, B 0.000, C 0.000 }
gfCNCPoint4[20385] = {X 338.2962, Y 62.6691, Z -6.3333, A 0.000, B 0.000, C 0.000 }
gfCNCPoint4[20386] = {X 337.7589, Y 64.2877, Z -6.3333, A 0.000, B 0.000, C 0.000 }
gfCNCPoint4[20387] = {X 337.0354, Y 65.8321, Z -6.3333, A 0.000, B 0.000, C 0.000 }
gfCNCPoint4[20388] = {X 336.1359, Y 67.2810, Z -6.3333, A 0.000, B 0.000, C 0.000 }
gfCNCPoint4[20389] = {X 335.0726, Y 68.6145, Z -6.3333, A 0.000, B 0.000, C 0.000 }
gfCNCPoint4[20390] = {X 335.0736, Y 79.5896, Z -6.3333, A 0.000, B 0.000, C 0.000 }
gfCNCPoint4[20391] = {X 335.9715, Y 79.6970, Z -6.3333, A 0.000, B 0.000, C 0.000 }
gfCNCPoint4[20392] = {X 336.8718, Y 79.7824, Z -6.3333, A 0.000, B 0.000, C 0.000 }
gfCNCPoint4[20393] = {X 340.9430, Y 80.0564, Z -6.3333, A 0.000, B 0.000, C 0.000 }
gfCNCPoint4[20394] = {X 345.0208, Y 80.1988, Z -6.3333, A 0.000, B 0.000, C 0.000 }
gfCNCPoint4[20395] = {X 349.1011, Y 80.2093, Z -6.3333, A 0.000, B 0.000, C 0.000 }
gfCNCPoint4[20396] = {X 352.9064, Y 80.1491, Z -6.3333, A 0.000, B 0.000, C 0.000 }
gfCNCPoint4[20397] = {X 356.7069, Y 79.9500, Z -6.3333, A 0.000, B 0.000, C 0.000 }
gfCNCPoint4[20398] = {X 360.4976, Y 79.6123, Z -6.3333, A 0.000, B 0.000, C 0.000 }
gfCNCPoint4[20399] = {X 360.7591, Y 79.5822, Z -6.3333, A 0.000, B 0.000, C 0.000 }
gfCNCPoint4[20400] = {X 360.7585, Y 68.6230, Z -6.3333, A 0.000, B 0.000, C 0.000 }
gfCNCPoint4[20401] = {X 359.7295, Y 67.3407, Z -6.3333, A 0.000, B 0.000, C 0.000 }
gfCNCPoint4[20402] = {X 358.8525, Y 65.9500, Z -6.3333, A 0.000, B 0.000, C 0.000 }
gfCNCPoint4[20403] = {X 358.1389, Y 64.4689, Z -6.3333, A 0.000, B 0.000, C 0.000 }
gfCNCPoint4[20404] = {X 357.5977, Y 62.9165, Z -6.3333, A 0.000, B 0.000, C 0.000 }
gfCNCPoint4[20405] = {X 357.2360, Y 61.3127, Z -6.3333, A 0.000, B 0.000, C 0.000 }
gfCNCPoint4[20406] = {X 357.0916, Y 60.1639, Z -6.3333, A 0.000, B 0.000, C 0.000 }
gfCNCPoint4[20407] = {X 357.0395, Y 59.0073, Z -6.3333, A 0.000, B 0.000, C 0.000 }
gfCNCPoint4[20408] = {X 357.0394, Y 58.6400, Z -6.3333, A 0.000, B 0.000, C 0.000 }
gfCNCPoint4[20409] = {X 355.6990, Y 59.0309, Z -6.3333, A 0.000, B 0.000, C 0.000 }
gfCNCPoint4[20410] = {X 354.3433, Y 59.3651, Z -6.3333, A 0.000, B 0.000, C 0.000 }
gfCNCPoint4[20411] = {X 351.8450, Y 59.8258, Z -6.3333, A 0.000, B 0.000, C 0.000 }
gfCNCPoint4[20412] = {X 349.3187, Y 60.0940, Z -6.3333, A 0.000, B 0.000, C 0.000 }
gfCNCPoint4[20413] = {X 349.1568, Y 57.6995, Z -6.3333, A 0.000, B 0.000, C 0.000 }
gfCNCPoint4[20414] = {X 348.1783, Y 57.7500, Z -6.3333, A 0.000, B 0.000, C 0.000 }
gfCNCPoint4[20415] = {X 347.1986, Y 57.7694, Z -6.3333, A 0.000, B 0.000, C 0.000 }
gfCNCPoint4[20416] = {X 344.5555, Y 57.7204, Z -6.3333, A 0.000, B 0.000, C 0.000 }
gfCNCPoint4[20417] = {X 341.9258, Y 57.4505, Z -6.3333, A 0.000, B 0.000, C 0.000 }
gfCNCPoint4[20418] = {X 339.3279, Y 56.9615, Z -6.3333, A 0.000, B 0.000, C 0.000 }
gfCNCPoint4[20419] = {X 337.7709, Y 56.5583, Z -6.3333, A 0.000, B 0.000, C 0.000 }
gfCNCPoint4[20420] = {X 336.2365, Y 56.0763, Z -6.3333, A 0.000, B 0.000, C 0.000 }
gfCNCPoint4[20421] = {X 336.3521, Y 57.0351, Z -6.3333, A 0.000, B 0.000, C 0.000 }
